LIN {X 0,Y 418.948,Z 202.65,A -85,B 0,C 180,E1 -10203.452,E2 -10203.452} C_VEL
LIN {X 0,Y 418.263,Z 200.109,A -85,B 0,C 180,E1 -10203.965,E2 -10203.965} C_VEL
LIN {X 0,Y 418.238,Z 200.015,A -85,B 0,C 180,E1 -10207.224,E2 -10207.224} C_VEL
LIN {X 0,Y 418.241,Z 199.978,A -85,B 0,C 180,E1 -10209.683,E2 -10209.683} C_VEL
LIN {X 0,Y 418.228,Z 200.013,A -85,B 0,C 180,E1 -10212.321,E2 -10212.321} C_VEL
LIN {X 0,Y 418.234,Z 200.009,A -85,B 0,C 180,E1 -10215.109,E2 -10215.109} C_VEL
LIN {X 0,Y 418.238,Z 200.002,A -85,B 0,C 180,E1 -10217.767,E2 -10217.767} C_VEL
LIN {X 0,Y 418.256,Z 200.011,A -85,B 0,C 180,E1 -10220.618,E2 -10220.618} C_VEL
LIN {X 0,Y 418.241,Z 200.01,A -85,B 0,C 180,E1 -10223.976,E2 -10223.976} C_VEL
LIN {X 0,Y 418.255,Z 199.993,A -85,B 0,C 180,E1 -10227.156,E2 -10227.156} C_VEL
LIN {X 0,Y 418.266,Z 200.006,A -85,B 0,C 180,E1 -10230.895,E2 -10230.895} C_VEL
LIN {X 0,Y 418.265,Z 199.989,A -85,B 0,C 180,E1 -10234.096,E2 -10234.096} C_VEL
LIN {X 0,Y 418.235,Z 200.01,A -85,B 0,C 180,E1 -10237.264,E2 -10237.264} C_VEL
LIN {X 0,Y 418.281,Z 200.008,A -85,B 0,C 180,E1 -10240.364,E2 -10240.364} C_VEL
LIN {X 0,Y 418.315,Z 199.999,A -85,B 0,C 180,E1 -10243.405,E2 -10243.405} C_VEL
LIN {X 0,Y 418.344,Z 199.994,A -85,B 0,C 180,E1 -10246.999,E2 -10246.999} C_VEL
LIN {X 0,Y 418.338,Z 199.995,A -85,B 0,C 180,E1 -10250.329,E2 -10250.329} C_VEL
LIN {X 0,Y 418.49,Z 199.98,A -85,B 0,C 180,E1 -10253.249,E2 -10253.249} C_VEL
LIN {X 0,Y 418.337,Z 199.993,A -85,B 0,C 180,E1 -10255.182,E2 -10255.182} C_VEL
LIN {X 0,Y 418.54,Z 199.968,A -85,B 0,C 180,E1 -10258.076,E2 -10258.076} C_VEL
LIN {X 0,Y 418.668,Z 199.959,A -85,B 0,C 180,E1 -10260,E2 -10260} C_VEL
LIN {X 0,Y 418.499,Z 199.974,A -85,B 0,C 180,E1 -10262.888,E2 -10262.888} C_VEL
LIN {X 0,Y 418.491,Z 199.977,A -85,B 0,C 180,E1 -10266.751,E2 -10266.751} C_VEL
LIN {X 0,Y 418.398,Z 199.988,A -85,B 0,C 180,E1 -10268.695,E2 -10268.695} C_VEL
LIN {X 0,Y 418.313,Z 199.997,A -85,B 0,C 180,E1 -10271.631,E2 -10271.631} C_VEL
LIN {X 0,Y 418.302,Z 200.003,A -85,B 0,C 180,E1 -10274.597,E2 -10274.597} C_VEL
LIN {X 0,Y 418.286,Z 200.007,A -85,B 0,C 180,E1 -10277.604,E2 -10277.604} C_VEL
LIN {X 0,Y 418.248,Z 200.005,A -85,B 0,C 180,E1 -10280.663,E2 -10280.663} C_VEL
LIN {X 0,Y 418.286,Z 200.001,A -85,B 0,C 180,E1 -10283.781,E2 -10283.781} C_VEL
LIN {X 0,Y 418.309,Z 199.995,A -85,B 0,C 180,E1 -10287.071,E2 -10287.071} C_VEL
LIN {X 0,Y 418.243,Z 200.002,A -85,B 0,C 180,E1 -10290.272,E2 -10290.272} C_VEL
LIN {X 0,Y 418.248,Z 200.002,A -85,B 0,C 180,E1 -10293.677,E2 -10293.677} C_VEL
LIN {X 0,Y 418.245,Z 200.012,A -85,B 0,C 180,E1 -10297.224,E2 -10297.224} C_VEL
LIN {X 0,Y 418.245,Z 199.997,A -85,B 0,C 180,E1 -10299.683,E2 -10299.683} C_VEL
LIN {X 0,Y 418.229,Z 200.016,A -85,B 0,C 180,E1 -10302.321,E2 -10302.321} C_VEL
LIN {X 0,Y 418.236,Z 200.01,A -85,B 0,C 180,E1 -10305.109,E2 -10305.109} C_VEL
LIN {X 0,Y 418.241,Z 200.003,A -85,B 0,C 180,E1 -10307.767,E2 -10307.767} C_VEL
LIN {X 0,Y 418.257,Z 200.007,A -85,B 0,C 180,E1 -10311.559,E2 -10311.559} C_VEL
LIN {X 0,Y 418.261,Z 200.008,A -85,B 0,C 180,E1 -10315.159,E2 -10315.159} C_VEL
LIN {X 0,Y 418.264,Z 200.161,A -85,B 0,C 180,E1 -10317.936,E2 -10317.936} C_VEL
LIN {X 0,Y 421.61,Z 212.936,A -85,B 0,C 180,E1 -10320.666,E2 -10320.666} C_VEL
LIN {X 0,Y 424.492,Z 225.433,A -85,B 0,C 180,E1 -10323.183,E2 -10323.183} C_VEL
LIN {X 0,Y 424.056,Z 232.827,A -85,B 0,C 180,E1 -10324.475,E2 -10324.475} C_VEL
LIN {X 0,Y 423.178,Z 244.55,A -85,B 0,C 180,E1 -10326.446,E2 -10326.446} C_VEL
LIN {X 0,Y 428.61,Z 271.164,A -85,B 0,C 180,E1 -10327.259,E2 -10327.259} C_VEL
LIN {X 0,Y 427.159,Z 386.676,A -85,B 0,C 180,E1 -10329.126,E2 -10329.126} C_VEL
LIN {X 0,Y 426.648,Z 400.992,A -85,B 0,C 180,E1 -10329.541,E2 -10329.541} C_VEL
LIN {X 0,Y 426.043,Z 413.972,A -85,B 0,C 180,E1 -10330.098,E2 -10330.098} C_VEL
LIN {X 0,Y 425.195,Z 426.696,A -85,B 0,C 180,E1 -10330.821,E2 -10330.821} C_VEL
LIN {X 0,Y 424.185,Z 439.707,A -85,B 0,C 180,E1 -10331.776,E2 -10331.776} C_VEL
LIN {X 0,Y 423.012,Z 451.477,A -85,B 0,C 180,E1 -10332.848,E2 -10332.848} C_VEL
LIN {X 0,Y 422.014,Z 462.206,A -85,B 0,C 180,E1 -10334.051,E2 -10334.051} C_VEL
LIN {X 0,Y 421.84,Z 463.782,A -85,B 0,C 180,E1 -10334.248,E2 -10334.248} C_VEL
LIN {X 0,Y 420.765,Z 468.085,A -85,B 0,C 180,E1 -10334.781,E2 -10334.781} C_VEL
LIN {X 0,Y 417.353,Z 474.899,A -85,B 0,C 180,E1 -10335.649,E2 -10335.649} C_VEL
LIN {X 0,Y 413.895,Z 481.189,A -85,B 0,C 180,E1 -10336.592,E2 -10336.592} C_VEL
LIN {X 0,Y 412.765,Z 484.669,A -85,B 0,C 180,E1 -10337.236,E2 -10337.236} C_VEL
LIN {X 0,Y 411.874,Z 492.436,A -85,B 0,C 180,E1 -10338.932,E2 -10338.932} C_VEL
LIN {X 0,Y 411.196,Z 498.815,A -85,B 0,C 180,E1 -10340.655,E2 -10340.655} C_VEL
LIN {X 0,Y 410.701,Z 504.611,A -85,B 0,C 180,E1 -10342.675,E2 -10342.675} C_VEL
LIN {X 0,Y 410.463,Z 507.781,A -85,B 0,C 180,E1 -10344.103,E2 -10344.103} C_VEL
LIN {X 0,Y 410.21,Z 510.948,A -85,B 0,C 180,E1 -10346.07,E2 -10346.07} C_VEL
LIN {X 0,Y 410.075,Z 512.822,A -85,B 0,C 180,E1 -10348.035,E2 -10348.035} C_VEL
LIN {X 0,Y 409.976,Z 513.463,A -85,B 0,C 180,E1 -10350,E2 -10350} C_VEL
LIN {X 0,Y 410.065,Z 512.885,A -85,B 0,C 180,E1 -10351.964,E2 -10351.964} C_VEL
LIN {X 0,Y 410.187,Z 511.079,A -85,B 0,C 180,E1 -10353.929,E2 -10353.929} C_VEL
LIN {X 0,Y 410.456,Z 507.979,A -85,B 0,C 180,E1 -10355.896,E2 -10355.896} C_VEL
LIN {X 0,Y 410.733,Z 503.489,A -85,B 0,C 180,E1 -10357.867,E2 -10357.867} C_VEL
LIN {X 0,Y 411.326,Z 497.457,A -85,B 0,C 180,E1 -10359.837,E2 -10359.837} C_VEL
LIN {X 0,Y 412.044,Z 490.753,A -85,B 0,C 180,E1 -10361.561,E2 -10361.561} C_VEL
LIN {X 0,Y 413.022,Z 482.453,A -85,B 0,C 180,E1 -10363.28,E2 -10363.28} C_VEL
LIN {X 0,Y 413.928,Z 473.814,A -85,B 0,C 180,E1 -10364.754,E2 -10364.754} C_VEL
LIN {X 0,Y 415.113,Z 463.352,A -85,B 0,C 180,E1 -10366.221,E2 -10366.221} C_VEL
LIN {X 0,Y 416.199,Z 452.792,A -85,B 0,C 180,E1 -10367.441,E2 -10367.441} C_VEL
LIN {X 0,Y 417.416,Z 441.262,A -85,B 0,C 180,E1 -10368.529,E2 -10368.529} C_VEL
LIN {X 0,Y 418.401,Z 428.579,A -85,B 0,C 180,E1 -10369.502,E2 -10369.502} C_VEL
LIN {X 0,Y 419.385,Z 414.919,A -85,B 0,C 180,E1 -10370.31,E2 -10370.31} C_VEL
LIN {X 0,Y 420.082,Z 401.003,A -85,B 0,C 180,E1 -10370.92,E2 -10370.92} C_VEL
LIN {X 0,Y 420.614,Z 386.556,A -85,B 0,C 180,E1 -10371.342,E2 -10371.342} C_VEL
LIN {X 0,Y 422.183,Z 272.349,A -85,B 0,C 180,E1 -10373.21,E2 -10373.21} C_VEL
LIN {X 0,Y 416.52,Z 244.696,A -85,B 0,C 180,E1 -10374.076,E2 -10374.076} C_VEL
LIN {X 0,Y 416.759,Z 240.683,A -85,B 0,C 180,E1 -10374.716,E2 -10374.716} C_VEL
LIN {X 0,Y 417.817,Z 228.064,A -85,B 0,C 180,E1 -10376.937,E2 -10376.937} C_VEL
LIN {X 0,Y 414.837,Z 214.884,A -85,B 0,C 180,E1 -10379.622,E2 -10379.622} C_VEL
LIN {X 0,Y 411.239,Z 201.027,A -85,B 0,C 180,E1 -10382.638,E2 -10382.638} C_VEL
LIN {X 0,Y 411.198,Z 200.892,A -85,B 0,C 180,E1 -10385.528,E2 -10385.528} C_VEL
LIN {X 0,Y 411.216,Z 200.882,A -85,B 0,C 180,E1 -10389.223,E2 -10389.223} C_VEL
LIN {X 0,Y 411.179,Z 200.884,A -85,B 0,C 180,E1 -10392.695,E2 -10392.695} C_VEL
LIN {X 0,Y 411.165,Z 200.884,A -85,B 0,C 180,E1 -10395.88,E2 -10395.88} C_VEL
LIN {X 0,Y 411.16,Z 200.895,A -85,B 0,C 180,E1 -10398.771,E2 -10398.771} C_VEL
LIN {X 0,Y 411.192,Z 200.891,A -85,B 0,C 180,E1 -10402.026,E2 -10402.026} C_VEL
LIN {X 0,Y 411.201,Z 200.874,A -85,B 0,C 180,E1 -10405.666,E2 -10405.666} C_VEL
LIN {X 0,Y 411.193,Z 200.887,A -85,B 0,C 180,E1 -10409.152,E2 -10409.152} C_VEL
LIN {X 0,Y 411.254,Z 200.868,A -85,B 0,C 180,E1 -10412.522,E2 -10412.522} C_VEL
LIN {X 0,Y 411.221,Z 200.881,A -85,B 0,C 180,E1 -10415.784,E2 -10415.784} C_VEL
LIN {X 0,Y 411.19,Z 200.889,A -85,B 0,C 180,E1 -10418.965,E2 -10418.965} C_VEL
LIN {X 0,Y 411.246,Z 200.881,A -85,B 0,C 180,E1 -10422.084,E2 -10422.084} C_VEL
LIN {X 0,Y 411.256,Z 200.883,A -85,B 0,C 180,E1 -10425.147,E2 -10425.147} C_VEL
LIN {X 0,Y 411.277,Z 200.873,A -85,B 0,C 180,E1 -10428.167,E2 -10428.167} C_VEL
LIN {X 0,Y 411.475,Z 200.85,A -85,B 0,C 180,E1 -10432.146,E2 -10432.146} C_VEL
LIN {X 0,Y 411.468,Z 200.854,A -85,B 0,C 180,E1 -10434.118,E2 -10434.118} C_VEL
LIN {X 0,Y 411.507,Z 200.847,A -85,B 0,C 180,E1 -10438.042,E2 -10438.042} C_VEL
LIN {X 0,Y 411.635,Z 200.835,A -85,B 0,C 180,E1 -10440,E2 -10440} C_VEL
LIN {X 0,Y 411.459,Z 200.855,A -85,B 0,C 180,E1 -10442.937,E2 -10442.937} C_VEL
LIN {X 0,Y 411.453,Z 200.856,A -85,B 0,C 180,E1 -10446.867,E2 -10446.867} C_VEL
LIN {X 0,Y 411.286,Z 200.873,A -85,B 0,C 180,E1 -10449.839,E2 -10449.839} C_VEL
LIN {X 0,Y 411.298,Z 200.872,A -85,B 0,C 180,E1 -10453.104,E2 -10453.104} C_VEL
LIN {X 0,Y 411.25,Z 200.878,A -85,B 0,C 180,E1 -10456.889,E2 -10456.889} C_VEL
LIN {X 0,Y 411.223,Z 200.887,A -85,B 0,C 180,E1 -10459.987,E2 -10459.987} C_VEL
LIN {X 0,Y 411.196,Z 200.888,A -85,B 0,C 180,E1 -10463.148,E2 -10463.148} C_VEL
LIN {X 0,Y 411.231,Z 200.862,A -85,B 0,C 180,E1 -10466.381,E2 -10466.381} C_VEL
LIN {X 0,Y 411.194,Z 200.893,A -85,B 0,C 180,E1 -10469.713,E2 -10469.713} C_VEL
LIN {X 0,Y 411.2,Z 200.872,A -85,B 0,C 180,E1 -10473.156,E2 -10473.156} C_VEL
LIN {X 0,Y 411.187,Z 200.885,A -85,B 0,C 180,E1 -10476.553,E2 -10476.553} C_VEL
LIN {X 0,Y 411.212,Z 200.89,A -85,B 0,C 180,E1 -10479.729,E2 -10479.729} C_VEL
LIN {X 0,Y 411.168,Z 200.889,A -85,B 0,C 180,E1 -10483.134,E2 -10483.134} C_VEL
LIN {X 0,Y 411.163,Z 200.887,A -85,B 0,C 180,E1 -10485.882,E2 -10485.882} C_VEL
LIN {X 0,Y 411.158,Z 200.874,A -85,B 0,C 180,E1 -10488.772,E2 -10488.772} C_VEL
LIN {X 0,Y 411.186,Z 200.884,A -85,B 0,C 180,E1 -10492.026,E2 -10492.026} C_VEL
LIN {X 0,Y 411.246,Z 201.009,A -85,B 0,C 180,E1 -10495.536,E2 -10495.536} C_VEL
LIN {X 0,Y 415.16,Z 214.888,A -85,B 0,C 180,E1 -10498.206,E2 -10498.206} C_VEL
LIN {X 0,Y 418.193,Z 226.388,A -85,B 0,C 180,E1 -10500.281,E2 -10500.281} C_VEL
LIN {X 0,Y 419.41,Z 231.713,A -85,B 0,C 180,E1 -10501.2,E2 -10501.2} C_VEL
LIN {X 0,Y 418.207,Z 245.027,A -85,B 0,C 180,E1 -10503.147,E2 -10503.147} C_VEL
LIN {X 0,Y 422.74,Z 272.159,A -85,B 0,C 180,E1 -10503.981,E2 -10503.981} C_VEL
LIN {X 0,Y 420.155,Z 407.504,A -85,B 0,C 180,E1 -10506.463,E2 -10506.463} C_VEL
LIN {X 0,Y 419.399,Z 423.23,A -85,B 0,C 180,E1 -10506.94,E2 -10506.94} C_VEL
LIN {X 0,Y 418.546,Z 437.915,A -85,B 0,C 180,E1 -10507.585,E2 -10507.585} C_VEL
LIN {X 0,Y 417.477,Z 451.995,A -85,B 0,C 180,E1 -10508.393,E2 -10508.393} C_VEL
LIN {X 0,Y 416.343,Z 465.452,A -85,B 0,C 180,E1 -10509.368,E2 -10509.368} C_VEL
LIN {X 0,Y 415.216,Z 477.877,A -85,B 0,C 180,E1 -10510.471,E2 -10510.471} C_VEL
LIN {X 0,Y 414.074,Z 490.391,A -85,B 0,C 180,E1 -10511.811,E2 -10511.811} C_VEL
LIN {X 0,Y 413.093,Z 501.14,A -85,B 0,C 180,E1 -10513.189,E2 -10513.189} C_VEL
LIN {X 0,Y 412.123,Z 510.953,A -85,B 0,C 180,E1 -10514.674,E2 -10514.674} C_VEL
LIN {X 0,Y 411.31,Z 520.71,A -85,B 0,C 180,E1 -10516.437,E2 -10516.437} C_VEL
LIN {X 0,Y 410.753,Z 528.58,A -85,B 0,C 180,E1 -10518.152,E2 -10518.152} C_VEL
LIN {X 0,Y 410.429,Z 534.358,A -85,B 0,C 180,E1 -10519.643,E2 -10519.643} C_VEL
LIN {X 0,Y 410.127,Z 540.599,A -85,B 0,C 180,E1 -10521.625,E2 -10521.625} C_VEL
LIN {X 0,Y 410.046,Z 544.283,A -85,B 0,C 180,E1 -10523.11,E2 -10523.11} C_VEL
LIN {X 0,Y 409.971,Z 548.051,A -85,B 0,C 180,E1 -10525.083,E2 -10525.083} C_VEL
LIN {X 0,Y 409.984,Z 550.533,A -85,B 0,C 180,E1 -10527.053,E2 -10527.053} C_VEL
LIN {X 0,Y 409.975,Z 551.778,A -85,B 0,C 180,E1 -10529.018,E2 -10529.018} C_VEL
LIN {X 0,Y 409.976,Z 551.776,A -85,B 0,C 180,E1 -10530.983,E2 -10530.983} C_VEL
LIN {X 0,Y 409.985,Z 550.524,A -85,B 0,C 180,E1 -10532.948,E2 -10532.948} C_VEL
LIN {X 0,Y 410,Z 548.04,A -85,B 0,C 180,E1 -10534.917,E2 -10534.917} C_VEL
LIN {X 0,Y 410.067,Z 544.273,A -85,B 0,C 180,E1 -10536.891,E2 -10536.891} C_VEL
LIN {X 0,Y 410.193,Z 539.132,A -85,B 0,C 180,E1 -10538.871,E2 -10538.871} C_VEL
LIN {X 0,Y 410.542,Z 532.489,A -85,B 0,C 180,E1 -10540.854,E2 -10540.854} C_VEL
LIN {X 0,Y 411.093,Z 524.16,A -85,B 0,C 180,E1 -10542.841,E2 -10542.841} C_VEL
LIN {X 0,Y 411.781,Z 515.261,A -85,B 0,C 180,E1 -10544.581,E2 -10544.581} C_VEL
LIN {X 0,Y 412.706,Z 504.537,A -85,B 0,C 180,E1 -10546.319,E2 -10546.319} C_VEL
LIN {X 0,Y 413.76,Z 493.517,A -85,B 0,C 180,E1 -10547.803,E2 -10547.803} C_VEL
LIN {X 0,Y 414.841,Z 481.467,A -85,B 0,C 180,E1 -10549.162,E2 -10549.162} C_VEL
LIN {X 0,Y 415.92,Z 469.712,A -85,B 0,C 180,E1 -10550.267,E2 -10550.267} C_VEL
LIN {X 0,Y 417.161,Z 455.436,A -85,B 0,C 180,E1 -10551.366,E2 -10551.366} C_VEL
LIN {X 0,Y 418.232,Z 441.838,A -85,B 0,C 180,E1 -10552.2,E2 -10552.2} C_VEL
LIN {X 0,Y 419.174,Z 426.827,A -85,B 0,C 180,E1 -10552.911,E2 -10552.911} C_VEL
LIN {X 0,Y 419.925,Z 411.687,A -85,B 0,C 180,E1 -10553.421,E2 -10553.421} C_VEL
LIN {X 0,Y 420.517,Z 391.478,A -85,B 0,C 180,E1 -10553.844,E2 -10553.844} C_VEL
LIN {X 0,Y 422.719,Z 272.152,A -85,B 0,C 180,E1 -10556.011,E2 -10556.011} C_VEL
LIN {X 0,Y 418.252,Z 245.233,A -85,B 0,C 180,E1 -10556.826,E2 -10556.826} C_VEL
LIN {X 0,Y 419.408,Z 231.698,A -85,B 0,C 180,E1 -10558.801,E2 -10558.801} C_VEL
LIN {X 0,Y 416.321,Z 219.072,A -85,B 0,C 180,E1 -10561.021,E2 -10561.021} C_VEL
LIN {X 0,Y 412.289,Z 204.82,A -85,B 0,C 180,E1 -10563.681,E2 -10563.681} C_VEL
LIN {X 0,Y 411.246,Z 200.982,A -85,B 0,C 180,E1 -10564.465,E2 -10564.465} C_VEL
LIN {X 0,Y 411.198,Z 200.877,A -85,B 0,C 180,E1 -10568.168,E2 -10568.168} C_VEL
LIN {X 0,Y 411.162,Z 200.874,A -85,B 0,C 180,E1 -10571.228,E2 -10571.228} C_VEL
LIN {X 0,Y 411.174,Z 200.885,A -85,B 0,C 180,E1 -10574.49,E2 -10574.49} C_VEL
LIN {X 0,Y 411.175,Z 200.882,A -85,B 0,C 180,E1 -10578.195,E2 -10578.195} C_VEL
LIN {X 0,Y 411.22,Z 200.885,A -85,B 0,C 180,E1 -10580.776,E2 -10580.776} C_VEL
LIN {X 0,Y 411.196,Z 200.893,A -85,B 0,C 180,E1 -10584.471,E2 -10584.471} C_VEL
LIN {X 0,Y 411.205,Z 200.872,A -85,B 0,C 180,E1 -10586.873,E2 -10586.873} C_VEL
LIN {X 0,Y 411.231,Z 200.885,A -85,B 0,C 180,E1 -10590.644,E2 -10590.644} C_VEL
LIN {X 0,Y 411.234,Z 200.861,A -85,B 0,C 180,E1 -10593.619,E2 -10593.619} C_VEL
LIN {X 0,Y 411.2,Z 200.888,A -85,B 0,C 180,E1 -10596.852,E2 -10596.852} C_VEL
LIN {X 0,Y 411.213,Z 200.889,A -85,B 0,C 180,E1 -10600.05,E2 -10600.05} C_VEL
LIN {X 0,Y 411.261,Z 200.877,A -85,B 0,C 180,E1 -10603.131,E2 -10603.131} C_VEL
LIN {X 0,Y 411.303,Z 200.871,A -85,B 0,C 180,E1 -10606.896,E2 -10606.896} C_VEL
LIN {X 0,Y 411.29,Z 200.872,A -85,B 0,C 180,E1 -10610.161,E2 -10610.161} C_VEL
LIN {X 0,Y 411.454,Z 200.856,A -85,B 0,C 180,E1 -10613.133,E2 -10613.133} C_VEL
LIN {X 0,Y 411.308,Z 200.868,A -85,B 0,C 180,E1 -10615.099,E2 -10615.099} C_VEL
LIN {X 0,Y 411.509,Z 200.844,A -85,B 0,C 180,E1 -10618.043,E2 -10618.043} C_VEL
LIN {X 0,Y 411.637,Z 200.835,A -85,B 0,C 180,E1 -10620,E2 -10620} C_VEL
LIN {X 0,Y 411.456,Z 200.852,A -85,B 0,C 180,E1 -10622.937,E2 -10622.937} C_VEL
LIN {X 0,Y 411.458,Z 200.854,A -85,B 0,C 180,E1 -10626.867,E2 -10626.867} C_VEL
LIN {X 0,Y 411.352,Z 200.866,A -85,B 0,C 180,E1 -10628.845,E2 -10628.845} C_VEL
LIN {X 0,Y 411.282,Z 200.872,A -85,B 0,C 180,E1 -10631.833,E2 -10631.833} C_VEL
LIN {X 0,Y 411.259,Z 200.882,A -85,B 0,C 180,E1 -10634.853,E2 -10634.853} C_VEL
LIN {X 0,Y 411.251,Z 200.881,A -85,B 0,C 180,E1 -10637.915,E2 -10637.915} C_VEL
LIN {X 0,Y 411.195,Z 200.888,A -85,B 0,C 180,E1 -10641.034,E2 -10641.034} C_VEL
LIN {X 0,Y 411.225,Z 200.88,A -85,B 0,C 180,E1 -10644.216,E2 -10644.216} C_VEL
LIN {X 0,Y 411.258,Z 200.868,A -85,B 0,C 180,E1 -10647.478,E2 -10647.478} C_VEL
LIN {X 0,Y 411.188,Z 200.886,A -85,B 0,C 180,E1 -10650.848,E2 -10650.848} C_VEL
LIN {X 0,Y 411.206,Z 200.874,A -85,B 0,C 180,E1 -10654.334,E2 -10654.334} C_VEL
LIN {X 0,Y 411.196,Z 200.889,A -85,B 0,C 180,E1 -10657.974,E2 -10657.974} C_VEL
LIN {X 0,Y 411.164,Z 200.893,A -85,B 0,C 180,E1 -10661.229,E2 -10661.229} C_VEL
LIN {X 0,Y 411.176,Z 200.883,A -85,B 0,C 180,E1 -10664.491,E2 -10664.491} C_VEL
LIN {X 0,Y 411.178,Z 200.884,A -85,B 0,C 180,E1 -10668.195,E2 -10668.195} C_VEL
LIN {X 0,Y 411.22,Z 200.881,A -85,B 0,C 180,E1 -10670.776,E2 -10670.776} C_VEL
LIN {X 0,Y 411.2,Z 200.891,A -85,B 0,C 180,E1 -10674.472,E2 -10674.472} C_VEL
LIN {X 0,Y 411.231,Z 201.077,A -85,B 0,C 180,E1 -10677.484,E2 -10677.484} C_VEL
LIN {X 0,Y 414.151,Z 212.297,A -85,B 0,C 180,E1 -10679.935,E2 -10679.935} C_VEL
LIN {X 0,Y 416.984,Z 224.123,A -85,B 0,C 180,E1 -10682.387,E2 -10682.387} C_VEL
LIN {X 0,Y 417.795,Z 228.696,A -85,B 0,C 180,E1 -10683.289,E2 -10683.289} C_VEL
LIN {X 0,Y 416.48,Z 244.569,A -85,B 0,C 180,E1 -10686.016,E2 -10686.016} C_VEL
LIN {X 0,Y 422.058,Z 271.648,A -85,B 0,C 180,E1 -10686.867,E2 -10686.867} C_VEL
LIN {X 0,Y 420.622,Z 386.454,A -85,B 0,C 180,E1 -10688.754,E2 -10688.754} C_VEL
LIN {X 0,Y 420.091,Z 400.957,A -85,B 0,C 180,E1 -10689.175,E2 -10689.175} C_VEL
LIN {X 0,Y 419.399,Z 414.888,A -85,B 0,C 180,E1 -10689.787,E2 -10689.787} C_VEL
LIN {X 0,Y 418.519,Z 427.216,A -85,B 0,C 180,E1 -10690.503,E2 -10690.503} C_VEL
LIN {X 0,Y 417.473,Z 440.174,A -85,B 0,C 180,E1 -10691.473,E2 -10691.473} C_VEL
LIN {X 0,Y 416.257,Z 451.907,A -85,B 0,C 180,E1 -10692.561,E2 -10692.561} C_VEL
LIN {X 0,Y 415.192,Z 462.612,A -85,B 0,C 180,E1 -10693.782,E2 -10693.782} C_VEL
LIN {X 0,Y 413.989,Z 473.195,A -85,B 0,C 180,E1 -10695.247,E2 -10695.247} C_VEL
LIN {X 0,Y 413.118,Z 481.937,A -85,B 0,C 180,E1 -10696.723,E2 -10696.723} C_VEL
LIN {X 0,Y 412.765,Z 484.669,A -85,B 0,C 180,E1 -10697.236,E2 -10697.236} C_VEL
LIN {X 0,Y 411.645,Z 488.055,A -85,B 0,C 180,E1 -10697.901,E2 -10697.901} C_VEL
LIN {X 0,Y 408.234,Z 493.211,A -85,B 0,C 180,E1 -10698.985,E2 -10698.985} C_VEL
LIN {X 0,Y 404.961,Z 497.856,A -85,B 0,C 180,E1 -10700.126,E2 -10700.126} C_VEL
LIN {X 0,Y 404.063,Z 500.337,A -85,B 0,C 180,E1 -10700.87,E2 -10700.87} C_VEL
LIN {X 0,Y 403.663,Z 504.834,A -85,B 0,C 180,E1 -10702.497,E2 -10702.497} C_VEL
LIN {X 0,Y 403.421,Z 508.12,A -85,B 0,C 180,E1 -10704,E2 -10704} C_VEL
LIN {X 0,Y 403.121,Z 511.284,A -85,B 0,C 180,E1 -10706.001,E2 -10706.001} C_VEL
LIN {X 0,Y 403.006,Z 513.154,A -85,B 0,C 180,E1 -10708.001,E2 -10708.001} C_VEL
LIN {X 0,Y 402.898,Z 513.795,A -85,B 0,C 180,E1 -10710,E2 -10710} C_VEL
LIN {X 0,Y 402.997,Z 513.217,A -85,B 0,C 180,E1 -10711.998,E2 -10711.998} C_VEL
LIN {X 0,Y 403.125,Z 512.467,A -85,B 0,C 180,E1 -10712.998,E2 -10712.998} C_VEL
LIN {X 0,Y 403.156,Z 510.035,A -85,B 0,C 180,E1 -10715,E2 -10715} C_VEL
LIN {X 0,Y 403.566,Z 506.254,A -85,B 0,C 180,E1 -10717.001,E2 -10717.001} C_VEL
LIN {X 0,Y 404.001,Z 501.021,A -85,B 0,C 180,E1 -10719.007,E2 -10719.007} C_VEL
LIN {X 0,Y 404.756,Z 494.15,A -85,B 0,C 180,E1 -10721.011,E2 -10721.011} C_VEL
LIN {X 0,Y 405.625,Z 486.583,A -85,B 0,C 180,E1 -10722.762,E2 -10722.762} C_VEL
LIN {X 0,Y 406.65,Z 477.932,A -85,B 0,C 180,E1 -10724.393,E2 -10724.393} C_VEL
LIN {X 0,Y 407.658,Z 469.228,A -85,B 0,C 180,E1 -10725.755,E2 -10725.755} C_VEL
LIN {X 0,Y 408.905,Z 458.721,A -85,B 0,C 180,E1 -10727.117,E2 -10727.117} C_VEL
LIN {X 0,Y 410.085,Z 447.116,A -85,B 0,C 180,E1 -10728.355,E2 -10728.355} C_VEL
LIN {X 0,Y 411.244,Z 435.757,A -85,B 0,C 180,E1 -10729.336,E2 -10729.336} C_VEL
LIN {X 0,Y 412.21,Z 423.673,A -85,B 0,C 180,E1 -10730.181,E2 -10730.181} C_VEL
LIN {X 0,Y 413.102,Z 409.749,A -85,B 0,C 180,E1 -10730.932,E2 -10730.932} C_VEL
LIN {X 0,Y 413.733,Z 396.35,A -85,B 0,C 180,E1 -10731.453,E2 -10731.453} C_VEL
LIN {X 0,Y 414.151,Z 383.076,A -85,B 0,C 180,E1 -10731.79,E2 -10731.79} C_VEL
LIN {X 0,Y 415.75,Z 273.499,A -85,B 0,C 180,E1 -10733.597,E2 -10733.597} C_VEL
LIN {X 0,Y 410.069,Z 245.992,A -85,B 0,C 180,E1 -10734.467,E2 -10734.467} C_VEL
LIN {X 0,Y 409.807,Z 244.124,A -85,B 0,C 180,E1 -10734.578,E2 -10734.578} C_VEL
LIN {X 0,Y 411.051,Z 230.507,A -85,B 0,C 180,E1 -10736.99,E2 -10736.99} C_VEL
LIN {X 0,Y 408.624,Z 219.018,A -85,B 0,C 180,E1 -10739.351,E2 -10739.351} C_VEL
LIN {X 0,Y 405.098,Z 205.35,A -85,B 0,C 180,E1 -10742.323,E2 -10742.323} C_VEL
LIN {X 0,Y 404.175,Z 201.859,A -85,B 0,C 180,E1 -10743.152,E2 -10743.152} C_VEL
LIN {X 0,Y 404.142,Z 201.763,A -85,B 0,C 180,E1 -10746.245,E2 -10746.245} C_VEL
LIN {X 0,Y 404.154,Z 201.763,A -85,B 0,C 180,E1 -10748.756,E2 -10748.756} C_VEL
LIN {X 0,Y 404.12,Z 201.766,A -85,B 0,C 180,E1 -10751.599,E2 -10751.599} C_VEL
LIN {X 0,Y 404.144,Z 201.767,A -85,B 0,C 180,E1 -10754.521,E2 -10754.521} C_VEL
LIN {X 0,Y 404.133,Z 201.768,A -85,B 0,C 180,E1 -10757.295,E2 -10757.295} C_VEL
LIN {X 0,Y 404.165,Z 201.751,A -85,B 0,C 180,E1 -10759.955,E2 -10759.955} C_VEL
LIN {X 0,Y 404.135,Z 201.772,A -85,B 0,C 180,E1 -10763.124,E2 -10763.124} C_VEL
LIN {X 0,Y 404.14,Z 201.758,A -85,B 0,C 180,E1 -10766.187,E2 -10766.187} C_VEL
LIN {X 0,Y 404.148,Z 201.758,A -85,B 0,C 180,E1 -10769.715,E2 -10769.715} C_VEL
LIN {X 0,Y 404.19,Z 201.754,A -85,B 0,C 180,E1 -10773.122,E2 -10773.122} C_VEL
LIN {X 0,Y 404.171,Z 201.762,A -85,B 0,C 180,E1 -10775.334,E2 -10775.334} C_VEL
LIN {X 0,Y 404.132,Z 201.77,A -85,B 0,C 180,E1 -10778.58,E2 -10778.58} C_VEL
LIN {X 0,Y 404.204,Z 201.758,A -85,B 0,C 180,E1 -10781.761,E2 -10781.761} C_VEL
LIN {X 0,Y 404.201,Z 201.758,A -85,B 0,C 180,E1 -10784.882,E2 -10784.882} C_VEL
LIN {X 0,Y 404.25,Z 201.748,A -85,B 0,C 180,E1 -10787.958,E2 -10787.958} C_VEL
LIN {X 0,Y 404.427,Z 201.728,A -85,B 0,C 180,E1 -10792.099,E2 -10792.099} C_VEL
LIN {X 0,Y 404.417,Z 201.731,A -85,B 0,C 180,E1 -10794.015,E2 -10794.015} C_VEL
LIN {X 0,Y 404.476,Z 201.722,A -85,B 0,C 180,E1 -10798.008,E2 -10798.008} C_VEL
LIN {X 0,Y 404.604,Z 201.711,A -85,B 0,C 180,E1 -10800,E2 -10800} C_VEL
LIN {X 0,Y 404.416,Z 201.733,A -85,B 0,C 180,E1 -10802.988,E2 -10802.988} C_VEL
LIN {X 0,Y 404.404,Z 201.734,A -85,B 0,C 180,E1 -10806.987,E2 -10806.987} C_VEL
LIN {X 0,Y 404.251,Z 201.749,A -85,B 0,C 180,E1 -10810.012,E2 -10810.012} C_VEL
LIN {X 0,Y 404.259,Z 201.748,A -85,B 0,C 180,E1 -10813.211,E2 -10813.211} C_VEL
LIN {X 0,Y 404.209,Z 201.755,A -85,B 0,C 180,E1 -10817.007,E2 -10817.007} C_VEL
LIN {X 0,Y 404.157,Z 201.763,A -85,B 0,C 180,E1 -10820.352,E2 -10820.352} C_VEL
LIN {X 0,Y 404.163,Z 201.768,A -85,B 0,C 180,E1 -10823.575,E2 -10823.575} C_VEL
LIN {X 0,Y 404.177,Z 201.744,A -85,B 0,C 180,E1 -10825.767,E2 -10825.767} C_VEL
LIN {X 0,Y 404.189,Z 201.752,A -85,B 0,C 180,E1 -10828,E2 -10828} C_VEL
LIN {X 0,Y 404.133,Z 201.756,A -85,B 0,C 180,E1 -10831.558,E2 -10831.558} C_VEL
LIN {X 0,Y 404.179,Z 201.763,A -85,B 0,C 180,E1 -10835.017,E2 -10835.017} C_VEL
LIN {X 0,Y 404.151,Z 201.761,A -85,B 0,C 180,E1 -10838.757,E2 -10838.757} C_VEL
LIN {X 0,Y 404.117,Z 201.761,A -85,B 0,C 180,E1 -10841.6,E2 -10841.6} C_VEL
LIN {X 0,Y 404.14,Z 201.768,A -85,B 0,C 180,E1 -10844.523,E2 -10844.523} C_VEL
LIN {X 0,Y 404.131,Z 201.773,A -85,B 0,C 180,E1 -10847.296,E2 -10847.296} C_VEL
LIN {X 0,Y 404.165,Z 201.73,A -85,B 0,C 180,E1 -10849.956,E2 -10849.956} C_VEL
LIN {X 0,Y 404.131,Z 201.765,A -85,B 0,C 180,E1 -10853.126,E2 -10853.126} C_VEL
LIN {X 0,Y 404.186,Z 201.933,A -85,B 0,C 180,E1 -10855.035,E2 -10855.035} C_VEL
LIN {X 0,Y 408.125,Z 215.592,A -85,B 0,C 180,E1 -10857.737,E2 -10857.737} C_VEL
LIN {X 0,Y 411.373,Z 227.977,A -85,B 0,C 180,E1 -10860.02,E2 -10860.02} C_VEL
LIN {X 0,Y 412.687,Z 233.627,A -85,B 0,C 180,E1 -10861.02,E2 -10861.02} C_VEL
LIN {X 0,Y 411.577,Z 245.037,A -85,B 0,C 180,E1 -10862.709,E2 -10862.709} C_VEL
LIN {X 0,Y 416.223,Z 272.495,A -85,B 0,C 180,E1 -10863.576,E2 -10863.576} C_VEL
LIN {X 0,Y 413.957,Z 393.97,A -85,B 0,C 180,E1 -10865.822,E2 -10865.822} C_VEL
LIN {X 0,Y 413.375,Z 412.135,A -85,B 0,C 180,E1 -10866.219,E2 -10866.219} C_VEL
LIN {X 0,Y 412.587,Z 427.051,A -85,B 0,C 180,E1 -10866.736,E2 -10866.736} C_VEL
LIN {X 0,Y 411.7,Z 440.535,A -85,B 0,C 180,E1 -10867.379,E2 -10867.379} C_VEL
LIN {X 0,Y 410.538,Z 455.044,A -85,B 0,C 180,E1 -10868.273,E2 -10868.273} C_VEL
LIN {X 0,Y 409.202,Z 469.332,A -85,B 0,C 180,E1 -10869.386,E2 -10869.386} C_VEL
LIN {X 0,Y 408.008,Z 482.292,A -85,B 0,C 180,E1 -10870.636,E2 -10870.636} C_VEL
LIN {X 0,Y 406.891,Z 493.161,A -85,B 0,C 180,E1 -10871.887,E2 -10871.887} C_VEL
LIN {X 0,Y 405.848,Z 504.196,A -85,B 0,C 180,E1 -10873.398,E2 -10873.398} C_VEL
LIN {X 0,Y 404.948,Z 513.533,A -85,B 0,C 180,E1 -10874.911,E2 -10874.911} C_VEL
LIN {X 0,Y 404.213,Z 521.735,A -85,B 0,C 180,E1 -10876.477,E2 -10876.477} C_VEL
LIN {X 0,Y 403.641,Z 530.289,A -85,B 0,C 180,E1 -10878.45,E2 -10878.45} C_VEL
LIN {X 0,Y 403.157,Z 537.319,A -85,B 0,C 180,E1 -10880.468,E2 -10880.468} C_VEL
LIN {X 0,Y 402.972,Z 542.826,A -85,B 0,C 180,E1 -10882.484,E2 -10882.484} C_VEL
LIN {X 0,Y 402.916,Z 545.994,A -85,B 0,C 180,E1 -10883.993,E2 -10883.993} C_VEL
LIN {X 0,Y 402.849,Z 549.113,A -85,B 0,C 180,E1 -10885.999,E2 -10885.999} C_VEL
LIN {X 0,Y 402.945,Z 550.978,A -85,B 0,C 180,E1 -10888.001,E2 -10888.001} C_VEL
LIN {X 0,Y 402.891,Z 551.606,A -85,B 0,C 180,E1 -10890,E2 -10890} C_VEL
LIN {X 0,Y 402.946,Z 550.972,A -85,B 0,C 180,E1 -10891.999,E2 -10891.999} C_VEL
LIN {X 0,Y 402.854,Z 549.1,A -85,B 0,C 180,E1 -10894.002,E2 -10894.002} C_VEL
LIN {X 0,Y 402.965,Z 545.983,A -85,B 0,C 180,E1 -10896.007,E2 -10896.007} C_VEL
LIN {X 0,Y 403.029,Z 541.536,A -85,B 0,C 180,E1 -10898.019,E2 -10898.019} C_VEL
LIN {X 0,Y 403.22,Z 535.652,A -85,B 0,C 180,E1 -10900.038,E2 -10900.038} C_VEL
LIN {X 0,Y 403.764,Z 528.189,A -85,B 0,C 180,E1 -10902.057,E2 -10902.057} C_VEL
LIN {X 0,Y 404.318,Z 520.302,A -85,B 0,C 180,E1 -10903.803,E2 -10903.803} C_VEL
LIN {X 0,Y 405.218,Z 510.529,A -85,B 0,C 180,E1 -10905.595,E2 -10905.595} C_VEL
LIN {X 0,Y 406.161,Z 500.684,A -85,B 0,C 180,E1 -10907.107,E2 -10907.107} C_VEL
LIN {X 0,Y 407.276,Z 488.972,A -85,B 0,C 180,E1 -10908.616,E2 -10908.616} C_VEL
LIN {X 0,Y 408.438,Z 477.355,A -85,B 0,C 180,E1 -10909.867,E2 -10909.867} C_VEL
LIN {X 0,Y 409.674,Z 464.868,A -85,B 0,C 180,E1 -10910.984,E2 -10910.984} C_VEL
LIN {X 0,Y 410.835,Z 451.333,A -85,B 0,C 180,E1 -10911.975,E2 -10911.975} C_VEL
LIN {X 0,Y 411.885,Z 437.239,A -85,B 0,C 180,E1 -10912.795,E2 -10912.795} C_VEL
LIN {X 0,Y 412.798,Z 422.296,A -85,B 0,C 180,E1 -10913.451,E2 -10913.451} C_VEL
LIN {X 0,Y 413.572,Z 407.375,A -85,B 0,C 180,E1 -10913.903,E2 -10913.903} C_VEL
LIN {X 0,Y 416.143,Z 281.51,A -85,B 0,C 180,E1 -10916.243,E2 -10916.243} C_VEL
LIN {X 0,Y 416.122,Z 272.091,A -85,B 0,C 180,E1 -10916.428,E2 -10916.428} C_VEL
LIN {X 0,Y 411.611,Z 245.018,A -85,B 0,C 180,E1 -10917.279,E2 -10917.279} C_VEL
LIN {X 0,Y 412.654,Z 233.604,A -85,B 0,C 180,E1 -10918.984,E2 -10918.984} C_VEL
LIN {X 0,Y 409.548,Z 220.88,A -85,B 0,C 180,E1 -10921.271,E2 -10921.271} C_VEL
LIN {X 0,Y 405.847,Z 207.701,A -85,B 0,C 180,E1 -10923.777,E2 -10923.777} C_VEL
LIN {X 0,Y 404.189,Z 201.889,A -85,B 0,C 180,E1 -10924.966,E2 -10924.966} C_VEL
LIN {X 0,Y 404.147,Z 201.741,A -85,B 0,C 180,E1 -10928.758,E2 -10928.758} C_VEL
LIN {X 0,Y 404.121,Z 201.758,A -85,B 0,C 180,E1 -10931.6,E2 -10931.6} C_VEL
LIN {X 0,Y 404.144,Z 201.76,A -85,B 0,C 180,E1 -10934.522,E2 -10934.522} C_VEL
LIN {X 0,Y 404.134,Z 201.761,A -85,B 0,C 180,E1 -10937.295,E2 -10937.295} C_VEL
LIN {X 0,Y 404.167,Z 201.766,A -85,B 0,C 180,E1 -10939.955,E2 -10939.955} C_VEL
LIN {X 0,Y 404.134,Z 201.762,A -85,B 0,C 180,E1 -10943.125,E2 -10943.125} C_VEL
LIN {X 0,Y 404.143,Z 201.761,A -85,B 0,C 180,E1 -10946.188,E2 -10946.188} C_VEL
LIN {X 0,Y 404.143,Z 201.765,A -85,B 0,C 180,E1 -10949.715,E2 -10949.715} C_VEL
LIN {X 0,Y 404.192,Z 201.739,A -85,B 0,C 180,E1 -10953.123,E2 -10953.123} C_VEL
LIN {X 0,Y 404.174,Z 201.757,A -85,B 0,C 180,E1 -10955.334,E2 -10955.334} C_VEL
LIN {X 0,Y 404.136,Z 201.765,A -85,B 0,C 180,E1 -10958.581,E2 -10958.581} C_VEL
LIN {X 0,Y 404.208,Z 201.757,A -85,B 0,C 180,E1 -10961.762,E2 -10961.762} C_VEL
LIN {X 0,Y 404.204,Z 201.757,A -85,B 0,C 180,E1 -10964.882,E2 -10964.882} C_VEL
LIN {X 0,Y 404.254,Z 201.757,A -85,B 0,C 180,E1 -10967.959,E2 -10967.959} C_VEL
LIN {X 0,Y 404.403,Z 201.737,A -85,B 0,C 180,E1 -10972.129,E2 -10972.129} C_VEL
LIN {X 0,Y 404.42,Z 201.727,A -85,B 0,C 180,E1 -10974.015,E2 -10974.015} C_VEL
LIN {X 0,Y 404.478,Z 201.72,A -85,B 0,C 180,E1 -10978.009,E2 -10978.009} C_VEL
LIN {X 0,Y 404.607,Z 201.711,A -85,B 0,C 180,E1 -10980,E2 -10980} C_VEL
LIN {X 0,Y 404.414,Z 201.729,A -85,B 0,C 180,E1 -10982.989,E2 -10982.989} C_VEL
LIN {X 0,Y 404.41,Z 201.732,A -85,B 0,C 180,E1 -10986.987,E2 -10986.987} C_VEL
LIN {X 0,Y 404.256,Z 201.752,A -85,B 0,C 180,E1 -10990.012,E2 -10990.012} C_VEL
LIN {X 0,Y 404.265,Z 201.752,A -85,B 0,C 180,E1 -10993.212,E2 -10993.212} C_VEL
LIN {X 0,Y 404.214,Z 201.755,A -85,B 0,C 180,E1 -10997.007,E2 -10997.007} C_VEL
LIN {X 0,Y 404.162,Z 201.758,A -85,B 0,C 180,E1 -11000.352,E2 -11000.352} C_VEL
LIN {X 0,Y 404.168,Z 201.76,A -85,B 0,C 180,E1 -11003.575,E2 -11003.575} C_VEL
LIN {X 0,Y 404.183,Z 201.761,A -85,B 0,C 180,E1 -11005.767,E2 -11005.767} C_VEL
LIN {X 0,Y 404.194,Z 201.745,A -85,B 0,C 180,E1 -11008,E2 -11008} C_VEL
LIN {X 0,Y 404.138,Z 201.768,A -85,B 0,C 180,E1 -11011.558,E2 -11011.558} C_VEL
LIN {X 0,Y 404.185,Z 201.747,A -85,B 0,C 180,E1 -11015.016,E2 -11015.016} C_VEL
LIN {X 0,Y 404.152,Z 201.759,A -85,B 0,C 180,E1 -11018.757,E2 -11018.757} C_VEL
LIN {X 0,Y 404.123,Z 201.77,A -85,B 0,C 180,E1 -11021.6,E2 -11021.6} C_VEL
LIN {X 0,Y 404.145,Z 201.758,A -85,B 0,C 180,E1 -11024.522,E2 -11024.522} C_VEL
LIN {X 0,Y 404.138,Z 201.761,A -85,B 0,C 180,E1 -11027.296,E2 -11027.296} C_VEL
LIN {X 0,Y 404.17,Z 201.765,A -85,B 0,C 180,E1 -11029.956,E2 -11029.956} C_VEL
LIN {X 0,Y 404.139,Z 201.763,A -85,B 0,C 180,E1 -11033.125,E2 -11033.125} C_VEL
LIN {X 0,Y 404.146,Z 201.746,A -85,B 0,C 180,E1 -11036.188,E2 -11036.188} C_VEL
LIN {X 0,Y 404.201,Z 202.023,A -85,B 0,C 180,E1 -11037.017,E2 -11037.017} C_VEL
LIN {X 0,Y 407.279,Z 213.756,A -85,B 0,C 180,E1 -11039.633,E2 -11039.633} C_VEL
LIN {X 0,Y 410.148,Z 225.739,A -85,B 0,C 180,E1 -11042.164,E2 -11042.164} C_VEL
LIN {X 0,Y 411.044,Z 230.041,A -85,B 0,C 180,E1 -11043.035,E2 -11043.035} C_VEL
LIN {X 0,Y 409.77,Z 244.317,A -85,B 0,C 180,E1 -11045.542,E2 -11045.542} C_VEL
LIN {X 0,Y 411.399,Z 252.155,A -85,B 0,C 180,E1 -11045.834,E2 -11045.834} C_VEL
LIN {X 0,Y 415.713,Z 273.707,A -85,B 0,C 180,E1 -11046.502,E2 -11046.502} C_VEL
LIN {X 0,Y 414.041,Z 387.55,A -85,B 0,C 180,E1 -11048.4,E2 -11048.4} C_VEL
LIN {X 0,Y 413.497,Z 401.69,A -85,B 0,C 180,E1 -11048.828,E2 -11048.828} C_VEL
LIN {X 0,Y 412.772,Z 415.769,A -85,B 0,C 180,E1 -11049.464,E2 -11049.464} C_VEL
LIN {X 0,Y 411.863,Z 427.731,A -85,B 0,C 180,E1 -11050.175,E2 -11050.175} C_VEL
LIN {X 0,Y 410.777,Z 440.638,A -85,B 0,C 180,E1 -11051.16,E2 -11051.16} C_VEL
LIN {X 0,Y 409.522,Z 452.334,A -85,B 0,C 180,E1 -11052.265,E2 -11052.265} C_VEL
LIN {X 0,Y 408.401,Z 463.014,A -85,B 0,C 180,E1 -11053.504,E2 -11053.504} C_VEL
LIN {X 0,Y 407.127,Z 473.579,A -85,B 0,C 180,E1 -11054.993,E2 -11054.993} C_VEL
LIN {X 0,Y 406.21,Z 482.307,A -85,B 0,C 180,E1 -11056.493,E2 -11056.493} C_VEL
LIN {X 0,Y 405.117,Z 490.685,A -85,B 0,C 180,E1 -11058.238,E2 -11058.238} C_VEL
LIN {X 0,Y 404.367,Z 497.461,A -85,B 0,C 180,E1 -11059.991,E2 -11059.991} C_VEL
LIN {X 0,Y 404.063,Z 500.337,A -85,B 0,C 180,E1 -11060.87,E2 -11060.87} C_VEL
LIN {X 0,Y 403.176,Z 502.672,A -85,B 0,C 180,E1 -11061.631,E2 -11061.631} C_VEL
LIN {X 0,Y 400.001,Z 506.149,A -85,B 0,C 180,E1 -11062.879,E2 -11062.879} C_VEL
LIN {X 0,Y 397.38,Z 508.484,A -85,B 0,C 180,E1 -11063.907,E2 -11063.907} C_VEL
LIN {X 0,Y 396.217,Z 509.925,A -85,B 0,C 180,E1 -11064.721,E2 -11064.721} C_VEL
LIN {X 0,Y 396.099,Z 510.335,A -85,B 0,C 180,E1 -11065,E2 -11065} C_VEL
LIN {X 0,Y 396.049,Z 512.707,A -85,B 0,C 180,E1 -11066.948,E2 -11066.948} C_VEL
LIN {X 0,Y 395.847,Z 513.961,A -85,B 0,C 180,E1 -11068.982,E2 -11068.982} C_VEL
LIN {X 0,Y 395.846,Z 513.99,A -85,B 0,C 180,E1 -11071.017,E2 -11071.017} C_VEL
LIN {X 0,Y 396.042,Z 512.8,A -85,B 0,C 180,E1 -11073.051,E2 -11073.051} C_VEL
LIN {X 0,Y 396.101,Z 510.369,A -85,B 0,C 180,E1 -11075.089,E2 -11075.089} C_VEL
LIN {X 0,Y 396.511,Z 506.594,A -85,B 0,C 180,E1 -11077.127,E2 -11077.127} C_VEL
LIN {X 0,Y 396.979,Z 501.365,A -85,B 0,C 180,E1 -11079.168,E2 -11079.168} C_VEL
LIN {X 0,Y 397.778,Z 494.501,A -85,B 0,C 180,E1 -11081.206,E2 -11081.206} C_VEL
LIN {X 0,Y 398.712,Z 486.941,A -85,B 0,C 180,E1 -11082.987,E2 -11082.987} C_VEL
LIN {X 0,Y 399.723,Z 478.705,A -85,B 0,C 180,E1 -11084.576,E2 -11084.576} C_VEL
LIN {X 0,Y 400.831,Z 469.613,A -85,B 0,C 180,E1 -11086.03,E2 -11086.03} C_VEL
LIN {X 0,Y 402.144,Z 459.125,A -85,B 0,C 180,E1 -11087.414,E2 -11087.414} C_VEL
LIN {X 0,Y 403.379,Z 447.548,A -85,B 0,C 180,E1 -11088.671,E2 -11088.671} C_VEL
LIN {X 0,Y 404.574,Z 436.229,A -85,B 0,C 180,E1 -11089.667,E2 -11089.667} C_VEL
LIN {X 0,Y 405.642,Z 423.476,A -85,B 0,C 180,E1 -11090.571,E2 -11090.571} C_VEL
LIN {X 0,Y 406.513,Z 410.38,A -85,B 0,C 180,E1 -11091.287,E2 -11091.287} C_VEL
LIN {X 0,Y 407.218,Z 396.226,A -85,B 0,C 180,E1 -11091.847,E2 -11091.847} C_VEL
LIN {X 0,Y 407.651,Z 382.731,A -85,B 0,C 180,E1 -11092.189,E2 -11092.189} C_VEL
LIN {X 0,Y 409.19,Z 273.689,A -85,B 0,C 180,E1 -11094.023,E2 -11094.023} C_VEL
LIN {X 0,Y 403.477,Z 246.244,A -85,B 0,C 180,E1 -11094.917,E2 -11094.917} C_VEL
LIN {X 0,Y 403.152,Z 244.085,A -85,B 0,C 180,E1 -11095.048,E2 -11095.048} C_VEL
LIN {X 0,Y 404.243,Z 231.847,A -85,B 0,C 180,E1 -11097.256,E2 -11097.256} C_VEL
LIN {X 0,Y 401.413,Z 219.141,A -85,B 0,C 180,E1 -11099.932,E2 -11099.932} C_VEL
LIN {X 0,Y 397.96,Z 205.821,A -85,B 0,C 180,E1 -11102.904,E2 -11102.904} C_VEL
LIN {X 0,Y 397.145,Z 202.723,A -85,B 0,C 180,E1 -11103.672,E2 -11103.672} C_VEL
LIN {X 0,Y 397.095,Z 202.643,A -85,B 0,C 180,E1 -11107.209,E2 -11107.209} C_VEL
LIN {X 0,Y 397.099,Z 202.647,A -85,B 0,C 180,E1 -11110.445,E2 -11110.445} C_VEL
LIN {X 0,Y 397.099,Z 202.646,A -85,B 0,C 180,E1 -11113.648,E2 -11113.648} C_VEL
LIN {X 0,Y 397.099,Z 202.638,A -85,B 0,C 180,E1 -11116.52,E2 -11116.52} C_VEL
LIN {X 0,Y 397.109,Z 202.63,A -85,B 0,C 180,E1 -11120.422,E2 -11120.422} C_VEL
LIN {X 0,Y 397.105,Z 202.637,A -85,B 0,C 180,E1 -11124.265,E2 -11124.265} C_VEL
LIN {X 0,Y 397.11,Z 202.635,A -85,B 0,C 180,E1 -11126.726,E2 -11126.726} C_VEL
LIN {X 0,Y 397.128,Z 202.628,A -85,B 0,C 180,E1 -11130.296,E2 -11130.296} C_VEL
LIN {X 0,Y 397.189,Z 202.62,A -85,B 0,C 180,E1 -11132.609,E2 -11132.609} C_VEL
LIN {X 0,Y 397.127,Z 202.636,A -85,B 0,C 180,E1 -11135.981,E2 -11135.981} C_VEL
LIN {X 0,Y 397.132,Z 202.634,A -85,B 0,C 180,E1 -11139.704,E2 -11139.704} C_VEL
LIN {X 0,Y 397.175,Z 202.635,A -85,B 0,C 180,E1 -11142.844,E2 -11142.844} C_VEL
LIN {X 0,Y 397.22,Z 202.632,A -85,B 0,C 180,E1 -11146.679,E2 -11146.679} C_VEL
LIN {X 0,Y 397.211,Z 202.629,A -85,B 0,C 180,E1 -11149.809,E2 -11149.809} C_VEL
LIN {X 0,Y 397.357,Z 202.609,A -85,B 0,C 180,E1 -11152.888,E2 -11152.888} C_VEL
LIN {X 0,Y 397.248,Z 202.626,A -85,B 0,C 180,E1 -11154.925,E2 -11154.925} C_VEL
LIN {X 0,Y 397.445,Z 202.598,A -85,B 0,C 180,E1 -11157.973,E2 -11157.973} C_VEL
LIN {X 0,Y 397.573,Z 202.586,A -85,B 0,C 180,E1 -11160,E2 -11160} C_VEL
LIN {X 0,Y 397.375,Z 202.61,A -85,B 0,C 180,E1 -11163.041,E2 -11163.041} C_VEL
LIN {X 0,Y 397.357,Z 202.611,A -85,B 0,C 180,E1 -11167.112,E2 -11167.112} C_VEL
LIN {X 0,Y 397.211,Z 202.627,A -85,B 0,C 180,E1 -11170.191,E2 -11170.191} C_VEL
LIN {X 0,Y 397.219,Z 202.626,A -85,B 0,C 180,E1 -11173.321,E2 -11173.321} C_VEL
LIN {X 0,Y 397.175,Z 202.631,A -85,B 0,C 180,E1 -11177.155,E2 -11177.155} C_VEL
LIN {X 0,Y 397.096,Z 202.641,A -85,B 0,C 180,E1 -11180.73,E2 -11180.73} C_VEL
LIN {X 0,Y 397.126,Z 202.639,A -85,B 0,C 180,E1 -11184.019,E2 -11184.019} C_VEL
LIN {X 0,Y 397.188,Z 202.614,A -85,B 0,C 180,E1 -11187.39,E2 -11187.39} C_VEL
LIN {X 0,Y 397.072,Z 202.646,A -85,B 0,C 180,E1 -11190.883,E2 -11190.883} C_VEL
LIN {X 0,Y 397.12,Z 202.641,A -85,B 0,C 180,E1 -11194.494,E2 -11194.494} C_VEL
LIN {X 0,Y 397.098,Z 202.636,A -85,B 0,C 180,E1 -11198.275,E2 -11198.275} C_VEL
LIN {X 0,Y 397.083,Z 202.644,A -85,B 0,C 180,E1 -11200.909,E2 -11200.909} C_VEL
LIN {X 0,Y 397.096,Z 202.648,A -85,B 0,C 180,E1 -11203.649,E2 -11203.649} C_VEL
LIN {X 0,Y 397.097,Z 202.643,A -85,B 0,C 180,E1 -11206.522,E2 -11206.522} C_VEL
LIN {X 0,Y 397.107,Z 202.608,A -85,B 0,C 180,E1 -11210.423,E2 -11210.423} C_VEL
LIN {X 0,Y 397.098,Z 202.631,A -85,B 0,C 180,E1 -11214.265,E2 -11214.265} C_VEL
LIN {X 0,Y 397.146,Z 202.931,A -85,B 0,C 180,E1 -11214.541,E2 -11214.541} C_VEL
LIN {X 0,Y 401.09,Z 216.342,A -85,B 0,C 180,E1 -11217.253,E2 -11217.253} C_VEL
LIN {X 0,Y 404.839,Z 230.684,A -85,B 0,C 180,E1 -11219.957,E2 -11219.957} C_VEL
LIN {X 0,Y 405.932,Z 235.424,A -85,B 0,C 180,E1 -11220.809,E2 -11220.809} C_VEL
LIN {X 0,Y 405.017,Z 245.196,A -85,B 0,C 180,E1 -11222.269,E2 -11222.269} C_VEL
LIN {X 0,Y 409.891,Z 274.319,A -85,B 0,C 180,E1 -11223.199,E2 -11223.199} C_VEL
LIN {X 0,Y 407.079,Z 405.226,A -85,B 0,C 180,E1 -11225.658,E2 -11225.658} C_VEL
LIN {X 0,Y 406.381,Z 420.855,A -85,B 0,C 180,E1 -11226.123,E2 -11226.123} C_VEL
LIN {X 0,Y 405.429,Z 435.259,A -85,B 0,C 180,E1 -11226.742,E2 -11226.742} C_VEL
LIN {X 0,Y 404.373,Z 448.945,A -85,B 0,C 180,E1 -11227.521,E2 -11227.521} C_VEL
LIN {X 0,Y 403.082,Z 462.894,A -85,B 0,C 180,E1 -11228.522,E2 -11228.522} C_VEL
LIN {X 0,Y 401.811,Z 475.678,A -85,B 0,C 180,E1 -11229.658,E2 -11229.658} C_VEL
LIN {X 0,Y 400.601,Z 487.53,A -85,B 0,C 180,E1 -11230.929,E2 -11230.929} C_VEL
LIN {X 0,Y 399.496,Z 498.633,A -85,B 0,C 180,E1 -11232.35,E2 -11232.35} C_VEL
LIN {X 0,Y 398.412,Z 508.67,A -85,B 0,C 180,E1 -11233.87,E2 -11233.87} C_VEL
LIN {X 0,Y 397.474,Z 518.581,A -85,B 0,C 180,E1 -11235.668,E2 -11235.668} C_VEL
LIN {X 0,Y 396.855,Z 526.012,A -85,B 0,C 180,E1 -11237.269,E2 -11237.269} C_VEL
LIN {X 0,Y 396.322,Z 533.657,A -85,B 0,C 180,E1 -11239.27,E2 -11239.27} C_VEL
LIN {X 0,Y 395.989,Z 539.911,A -85,B 0,C 180,E1 -11241.324,E2 -11241.324} C_VEL
LIN {X 0,Y 395.885,Z 543.602,A -85,B 0,C 180,E1 -11242.862,E2 -11242.862} C_VEL
LIN {X 0,Y 395.801,Z 547.378,A -85,B 0,C 180,E1 -11244.907,E2 -11244.907} C_VEL
LIN {X 0,Y 395.783,Z 549.865,A -85,B 0,C 180,E1 -11246.947,E2 -11246.947} C_VEL
LIN {X 0,Y 395.875,Z 550.646,A -85,B 0,C 180,E1 -11247.966,E2 -11247.966} C_VEL
LIN {X 0,Y 395.816,Z 551.274,A -85,B 0,C 180,E1 -11250,E2 -11250} C_VEL
LIN {X 0,Y 395.875,Z 550.64,A -85,B 0,C 180,E1 -11252.035,E2 -11252.035} C_VEL
LIN {X 0,Y 395.775,Z 548.765,A -85,B 0,C 180,E1 -11254.073,E2 -11254.073} C_VEL
LIN {X 0,Y 395.896,Z 545.455,A -85,B 0,C 180,E1 -11256.218,E2 -11256.218} C_VEL
LIN {X 0,Y 395.941,Z 541.19,A -85,B 0,C 180,E1 -11258.164,E2 -11258.164} C_VEL
LIN {X 0,Y 396.165,Z 535.3,A -85,B 0,C 180,E1 -11260.219,E2 -11260.219} C_VEL
LIN {X 0,Y 396.769,Z 527.83,A -85,B 0,C 180,E1 -11262.272,E2 -11262.272} C_VEL
LIN {X 0,Y 397.352,Z 519.805,A -85,B 0,C 180,E1 -11264.076,E2 -11264.076} C_VEL
LIN {X 0,Y 398.277,Z 510.145,A -85,B 0,C 180,E1 -11265.874,E2 -11265.874} C_VEL
LIN {X 0,Y 399.272,Z 500.284,A -85,B 0,C 180,E1 -11267.412,E2 -11267.412} C_VEL
LIN {X 0,Y 400.451,Z 488.55,A -85,B 0,C 180,E1 -11268.946,E2 -11268.946} C_VEL
LIN {X 0,Y 401.691,Z 476.904,A -85,B 0,C 180,E1 -11270.215,E2 -11270.215} C_VEL
LIN {X 0,Y 402.954,Z 464.375,A -85,B 0,C 180,E1 -11271.351,E2 -11271.351} C_VEL
LIN {X 0,Y 404.232,Z 450.789,A -85,B 0,C 180,E1 -11272.354,E2 -11272.354} C_VEL
LIN {X 0,Y 405.315,Z 436.776,A -85,B 0,C 180,E1 -11273.177,E2 -11273.177} C_VEL
LIN {X 0,Y 406.273,Z 421.498,A -85,B 0,C 180,E1 -11273.851,E2 -11273.851} C_VEL
LIN {X 0,Y 407.078,Z 406.249,A -85,B 0,C 180,E1 -11274.309,E2 -11274.309} C_VEL
LIN {X 0,Y 409.884,Z 274.359,A -85,B 0,C 180,E1 -11276.789,E2 -11276.789} C_VEL
LIN {X 0,Y 405.007,Z 245.16,A -85,B 0,C 180,E1 -11277.721,E2 -11277.721} C_VEL
LIN {X 0,Y 405.891,Z 235.392,A -85,B 0,C 180,E1 -11279.195,E2 -11279.195} C_VEL
LIN {X 0,Y 402.761,Z 222.47,A -85,B 0,C 180,E1 -11281.566,E2 -11281.566} C_VEL
LIN {X 0,Y 398.74,Z 208.285,A -85,B 0,C 180,E1 -11284.334,E2 -11284.334} C_VEL
LIN {X 0,Y 397.103,Z 202.778,A -85,B 0,C 180,E1 -11285.5,E2 -11285.5} C_VEL
LIN {X 0,Y 397.124,Z 202.613,A -85,B 0,C 180,E1 -11288.86,E2 -11288.86} C_VEL
LIN {X 0,Y 397.067,Z 202.649,A -85,B 0,C 180,E1 -11292.267,E2 -11292.267} C_VEL
LIN {X 0,Y 397.085,Z 202.642,A -85,B 0,C 180,E1 -11295.069,E2 -11295.069} C_VEL
LIN {X 0,Y 397.064,Z 202.638,A -85,B 0,C 180,E1 -11298.021,E2 -11298.021} C_VEL
LIN {X 0,Y 397.13,Z 202.637,A -85,B 0,C 180,E1 -11301.138,E2 -11301.138} C_VEL
LIN {X 0,Y 397.117,Z 202.647,A -85,B 0,C 180,E1 -11304.497,E2 -11304.497} C_VEL
LIN {X 0,Y 397.076,Z 202.63,A -85,B 0,C 180,E1 -11307.928,E2 -11307.928} C_VEL
LIN {X 0,Y 397.12,Z 202.639,A -85,B 0,C 180,E1 -11311.456,E2 -11311.456} C_VEL
LIN {X 0,Y 397.15,Z 202.622,A -85,B 0,C 180,E1 -11314.488,E2 -11314.488} C_VEL
LIN {X 0,Y 397.106,Z 202.643,A -85,B 0,C 180,E1 -11317.086,E2 -11317.086} C_VEL
LIN {X 0,Y 397.146,Z 202.641,A -85,B 0,C 180,E1 -11320.353,E2 -11320.353} C_VEL
LIN {X 0,Y 397.164,Z 202.635,A -85,B 0,C 180,E1 -11323.553,E2 -11323.553} C_VEL
LIN {X 0,Y 397.226,Z 202.625,A -85,B 0,C 180,E1 -11326.703,E2 -11326.703} C_VEL
LIN {X 0,Y 397.215,Z 202.626,A -85,B 0,C 180,E1 -11329.809,E2 -11329.809} C_VEL
LIN {X 0,Y 397.35,Z 202.612,A -85,B 0,C 180,E1 -11332.888,E2 -11332.888} C_VEL
LIN {X 0,Y 397.252,Z 202.618,A -85,B 0,C 180,E1 -11334.925,E2 -11334.925} C_VEL
LIN {X 0,Y 397.447,Z 202.596,A -85,B 0,C 180,E1 -11337.973,E2 -11337.973} C_VEL
LIN {X 0,Y 397.576,Z 202.586,A -85,B 0,C 180,E1 -11340,E2 -11340} C_VEL
LIN {X 0,Y 397.373,Z 202.605,A -85,B 0,C 180,E1 -11343.042,E2 -11343.042} C_VEL
LIN {X 0,Y 397.362,Z 202.609,A -85,B 0,C 180,E1 -11347.112,E2 -11347.112} C_VEL
LIN {X 0,Y 397.216,Z 202.629,A -85,B 0,C 180,E1 -11350.191,E2 -11350.191} C_VEL
LIN {X 0,Y 397.225,Z 202.63,A -85,B 0,C 180,E1 -11353.321,E2 -11353.321} C_VEL
LIN {X 0,Y 397.18,Z 202.633,A -85,B 0,C 180,E1 -11357.155,E2 -11357.155} C_VEL
LIN {X 0,Y 397.107,Z 202.639,A -85,B 0,C 180,E1 -11360.73,E2 -11360.73} C_VEL
LIN {X 0,Y 397.132,Z 202.636,A -85,B 0,C 180,E1 -11364.019,E2 -11364.019} C_VEL
LIN {X 0,Y 397.193,Z 202.62,A -85,B 0,C 180,E1 -11367.39,E2 -11367.39} C_VEL
LIN {X 0,Y 397.078,Z 202.644,A -85,B 0,C 180,E1 -11370.883,E2 -11370.883} C_VEL
LIN {X 0,Y 397.125,Z 202.626,A -85,B 0,C 180,E1 -11374.494,E2 -11374.494} C_VEL
LIN {X 0,Y 397.102,Z 202.645,A -85,B 0,C 180,E1 -11378.275,E2 -11378.275} C_VEL
LIN {X 0,Y 397.088,Z 202.639,A -85,B 0,C 180,E1 -11380.909,E2 -11380.909} C_VEL
LIN {X 0,Y 397.101,Z 202.637,A -85,B 0,C 180,E1 -11383.649,E2 -11383.649} C_VEL
LIN {X 0,Y 397.104,Z 202.644,A -85,B 0,C 180,E1 -11386.521,E2 -11386.521} C_VEL
LIN {X 0,Y 397.115,Z 202.638,A -85,B 0,C 180,E1 -11390.423,E2 -11390.423} C_VEL
LIN {X 0,Y 397.11,Z 202.643,A -85,B 0,C 180,E1 -11394.266,E2 -11394.266} C_VEL
LIN {X 0,Y 397.159,Z 202.787,A -85,B 0,C 180,E1 -11396.476,E2 -11396.476} C_VEL
LIN {X 0,Y 400.412,Z 215.228,A -85,B 0,C 180,E1 -11399.322,E2 -11399.322} C_VEL
LIN {X 0,Y 403.351,Z 227.373,A -85,B 0,C 180,E1 -11401.937,E2 -11401.937} C_VEL
LIN {X 0,Y 404.215,Z 231.384,A -85,B 0,C 180,E1 -11402.766,E2 -11402.766} C_VEL
LIN {X 0,Y 403.308,Z 242.106,A -85,B 0,C 180,E1 -11404.711,E2 -11404.711} C_VEL
LIN {X 0,Y 403.162,Z 244.79,A -85,B 0,C 180,E1 -11405.123,E2 -11405.123} C_VEL
LIN {X 0,Y 408.691,Z 271.445,A -85,B 0,C 180,E1 -11406.002,E2 -11406.002} C_VEL
LIN {X 0,Y 409.27,Z 274.688,A -85,B 0,C 180,E1 -11406.099,E2 -11406.099} C_VEL
LIN {X 0,Y 407.548,Z 387.361,A -85,B 0,C 180,E1 -11408.005,E2 -11408.005} C_VEL
LIN {X 0,Y 406.962,Z 401.646,A -85,B 0,C 180,E1 -11408.437,E2 -11408.437} C_VEL
LIN {X 0,Y 406.204,Z 415.769,A -85,B 0,C 180,E1 -11409.082,E2 -11409.082} C_VEL
LIN {X 0,Y 405.216,Z 428.243,A -85,B 0,C 180,E1 -11409.836,E2 -11409.836} C_VEL
LIN {X 0,Y 404.098,Z 441.097,A -85,B 0,C 180,E1 -11410.836,E2 -11410.836} C_VEL
LIN {X 0,Y 402.782,Z 452.76,A -85,B 0,C 180,E1 -11411.958,E2 -11411.958} C_VEL
LIN {X 0,Y 401.623,Z 463.413,A -85,B 0,C 180,E1 -11413.218,E2 -11413.218} C_VEL
LIN {X 0,Y 400.261,Z 473.963,A -85,B 0,C 180,E1 -11414.729,E2 -11414.729} C_VEL
LIN {X 0,Y 399.304,Z 482.676,A -85,B 0,C 180,E1 -11416.254,E2 -11416.254} C_VEL
LIN {X 0,Y 398.168,Z 491.043,A -85,B 0,C 180,E1 -11418.03,E2 -11418.03} C_VEL
LIN {X 0,Y 397.357,Z 497.812,A -85,B 0,C 180,E1 -11419.812,E2 -11419.812} C_VEL
LIN {X 0,Y 396.734,Z 503.91,A -85,B 0,C 180,E1 -11421.853,E2 -11421.853} C_VEL
LIN {X 0,Y 396.356,Z 508.459,A -85,B 0,C 180,E1 -11423.892,E2 -11423.892} C_VEL
LIN {X 0,Y 396.099,Z 510.335,A -85,B 0,C 180,E1 -11425,E2 -11425} C_VEL
LIN {X 0,Y 395.345,Z 511.534,A -85,B 0,C 180,E1 -11425.834,E2 -11425.834} C_VEL
LIN {X 0,Y 392.379,Z 513.098,A -85,B 0,C 180,E1 -11427.193,E2 -11427.193} C_VEL
LIN {X 0,Y 389.906,Z 513.952,A -85,B 0,C 180,E1 -11428.297,E2 -11428.297} C_VEL
LIN {X 0,Y 388.839,Z 514.332,A -85,B 0,C 180,E1 -11429.156,E2 -11429.156} C_VEL
LIN {X 0,Y 388.749,Z 514.37,A -85,B 0,C 180,E1 -11429.448,E2 -11429.448} C_VEL
LIN {X 0,Y 388.776,Z 514.322,A -85,B 0,C 180,E1 -11431.035,E2 -11431.035} C_VEL
LIN {X 0,Y 388.963,Z 513.133,A -85,B 0,C 180,E1 -11433.107,E2 -11433.107} C_VEL
LIN {X 0,Y 389.048,Z 510.704,A -85,B 0,C 180,E1 -11435.182,E2 -11435.182} C_VEL
LIN {X 0,Y 389.455,Z 506.933,A -85,B 0,C 180,E1 -11437.257,E2 -11437.257} C_VEL
LIN {X 0,Y 389.973,Z 501.708,A -85,B 0,C 180,E1 -11439.334,E2 -11439.334} C_VEL
LIN {X 0,Y 390.805,Z 494.85,A -85,B 0,C 180,E1 -11441.409,E2 -11441.409} C_VEL
LIN {X 0,Y 391.798,Z 487.298,A -85,B 0,C 180,E1 -11443.22,E2 -11443.22} C_VEL
LIN {X 0,Y 392.797,Z 479.487,A -85,B 0,C 180,E1 -11444.763,E2 -11444.763} C_VEL
LIN {X 0,Y 394.002,Z 469.997,A -85,B 0,C 180,E1 -11446.316,E2 -11446.316} C_VEL
LIN {X 0,Y 395.391,Z 459.528,A -85,B 0,C 180,E1 -11447.721,E2 -11447.721} C_VEL
LIN {X 0,Y 396.689,Z 447.976,A -85,B 0,C 180,E1 -11448.998,E2 -11448.998} C_VEL
LIN {X 0,Y 398.07,Z 435.13,A -85,B 0,C 180,E1 -11450.137,E2 -11450.137} C_VEL
LIN {X 0,Y 399.156,Z 422.492,A -85,B 0,C 180,E1 -11451.024,E2 -11451.024} C_VEL
LIN {X 0,Y 400.011,Z 409.698,A -85,B 0,C 180,E1 -11451.718,E2 -11451.718} C_VEL
LIN {X 0,Y 400.732,Z 396.095,A -85,B 0,C 180,E1 -11452.253,E2 -11452.253} C_VEL
LIN {X 0,Y 401.169,Z 382.381,A -85,B 0,C 180,E1 -11452.601,E2 -11452.601} C_VEL
LIN {X 0,Y 402.794,Z 274.93,A -85,B 0,C 180,E1 -11454.434,E2 -11454.434} C_VEL
LIN {X 0,Y 397.73,Z 250.174,A -85,B 0,C 180,E1 -11455.254,E2 -11455.254} C_VEL
LIN {X 0,Y 396.531,Z 244.414,A -85,B 0,C 180,E1 -11455.482,E2 -11455.482} C_VEL
LIN {X 0,Y 397.514,Z 234.03,A -85,B 0,C 180,E1 -11457.365,E2 -11457.365} C_VEL
LIN {X 0,Y 394.957,Z 222.226,A -85,B 0,C 180,E1 -11459.883,E2 -11459.883} C_VEL
LIN {X 0,Y 391.533,Z 208.955,A -85,B 0,C 180,E1 -11462.886,E2 -11462.886} C_VEL
LIN {X 0,Y 390.103,Z 203.638,A -85,B 0,C 180,E1 -11464.176,E2 -11464.176} C_VEL
LIN {X 0,Y 390.043,Z 203.528,A -85,B 0,C 180,E1 -11467.779,E2 -11467.779} C_VEL
LIN {X 0,Y 390.054,Z 203.525,A -85,B 0,C 180,E1 -11470.82,E2 -11470.82} C_VEL
LIN {X 0,Y 390.052,Z 203.526,A -85,B 0,C 180,E1 -11473.885,E2 -11473.885} C_VEL
LIN {X 0,Y 390.054,Z 203.517,A -85,B 0,C 180,E1 -11476.789,E2 -11476.789} C_VEL
LIN {X 0,Y 390.052,Z 203.511,A -85,B 0,C 180,E1 -11479.56,E2 -11479.56} C_VEL
LIN {X 0,Y 390.04,Z 203.525,A -85,B 0,C 180,E1 -11482.448,E2 -11482.448} C_VEL
LIN {X 0,Y 390.063,Z 203.507,A -85,B 0,C 180,E1 -11485.975,E2 -11485.975} C_VEL
LIN {X 0,Y 390.047,Z 203.513,A -85,B 0,C 180,E1 -11489.867,E2 -11489.867} C_VEL
LIN {X 0,Y 390.108,Z 203.509,A -85,B 0,C 180,E1 -11493.231,E2 -11493.231} C_VEL
LIN {X 0,Y 390.101,Z 203.512,A -85,B 0,C 180,E1 -11496.75,E2 -11496.75} C_VEL
LIN {X 0,Y 390.098,Z 203.51,A -85,B 0,C 180,E1 -11499.982,E2 -11499.982} C_VEL
LIN {X 0,Y 390.132,Z 203.507,A -85,B 0,C 180,E1 -11503.248,E2 -11503.248} C_VEL
LIN {X 0,Y 390.188,Z 203.509,A -85,B 0,C 180,E1 -11506.561,E2 -11506.561} C_VEL
LIN {X 0,Y 390.198,Z 203.506,A -85,B 0,C 180,E1 -11510.671,E2 -11510.671} C_VEL
LIN {X 0,Y 390.311,Z 203.486,A -85,B 0,C 180,E1 -11512.759,E2 -11512.759} C_VEL
LIN {X 0,Y 390.22,Z 203.502,A -85,B 0,C 180,E1 -11514.833,E2 -11514.833} C_VEL
LIN {X 0,Y 390.413,Z 203.473,A -85,B 0,C 180,E1 -11517.937,E2 -11517.937} C_VEL
LIN {X 0,Y 390.543,Z 203.462,A -85,B 0,C 180,E1 -11520,E2 -11520} C_VEL
LIN {X 0,Y 390.309,Z 203.49,A -85,B 0,C 180,E1 -11523.096,E2 -11523.096} C_VEL
LIN {X 0,Y 390.323,Z 203.484,A -85,B 0,C 180,E1 -11526.202,E2 -11526.202} C_VEL
LIN {X 0,Y 390.307,Z 203.491,A -85,B 0,C 180,E1 -11528.282,E2 -11528.282} C_VEL
LIN {X 0,Y 390.163,Z 203.507,A -85,B 0,C 180,E1 -11532.483,E2 -11532.483} C_VEL
LIN {X 0,Y 390.132,Z 203.513,A -85,B 0,C 180,E1 -11535.677,E2 -11535.677} C_VEL
LIN {X 0,Y 390.098,Z 203.514,A -85,B 0,C 180,E1 -11538.922,E2 -11538.922} C_VEL
LIN {X 0,Y 390.033,Z 203.525,A -85,B 0,C 180,E1 -11542.234,E2 -11542.234} C_VEL
LIN {X 0,Y 390.112,Z 203.495,A -85,B 0,C 180,E1 -11545.744,E2 -11545.744} C_VEL
LIN {X 0,Y 390.052,Z 203.521,A -85,B 0,C 180,E1 -11549.11,E2 -11549.11} C_VEL
LIN {X 0,Y 390.036,Z 203.504,A -85,B 0,C 180,E1 -11552.722,E2 -11552.722} C_VEL
LIN {X 0,Y 390.05,Z 203.521,A -85,B 0,C 180,E1 -11555.826,E2 -11555.826} C_VEL
LIN {X 0,Y 390.065,Z 203.519,A -85,B 0,C 180,E1 -11559.219,E2 -11559.219} C_VEL
LIN {X 0,Y 390.036,Z 203.514,A -85,B 0,C 180,E1 -11562.375,E2 -11562.375} C_VEL
LIN {X 0,Y 390.039,Z 203.516,A -85,B 0,C 180,E1 -11565.355,E2 -11565.355} C_VEL
LIN {X 0,Y 390.024,Z 203.517,A -85,B 0,C 180,E1 -11568.187,E2 -11568.187} C_VEL
LIN {X 0,Y 390.082,Z 203.486,A -85,B 0,C 180,E1 -11570.908,E2 -11570.908} C_VEL
LIN {X 0,Y 390.081,Z 203.67,A -85,B 0,C 180,E1 -11573.945,E2 -11573.945} C_VEL
LIN {X 0,Y 394.266,Z 217.866,A -85,B 0,C 180,E1 -11576.908,E2 -11576.908} C_VEL
LIN {X 0,Y 397.979,Z 232.03,A -85,B 0,C 180,E1 -11579.639,E2 -11579.639} C_VEL
LIN {X 0,Y 399.209,Z 238.195,A -85,B 0,C 180,E1 -11580.757,E2 -11580.757} C_VEL
LIN {X 0,Y 398.404,Z 245.126,A -85,B 0,C 180,E1 -11581.795,E2 -11581.795} C_VEL
LIN {X 0,Y 402.384,Z 268.468,A -85,B 0,C 180,E1 -11582.573,E2 -11582.573} C_VEL
LIN {X 0,Y 403.485,Z 275.824,A -85,B 0,C 180,E1 -11582.798,E2 -11582.798} C_VEL
LIN {X 0,Y 400.545,Z 405.523,A -85,B 0,C 180,E1 -11585.269,E2 -11585.269} C_VEL
LIN {X 0,Y 399.832,Z 420.969,A -85,B 0,C 180,E1 -11585.741,E2 -11585.741} C_VEL
LIN {X 0,Y 398.777,Z 436.145,A -85,B 0,C 180,E1 -11586.411,E2 -11586.411} C_VEL
LIN {X 0,Y 397.612,Z 450.404,A -85,B 0,C 180,E1 -11587.254,E2 -11587.254} C_VEL
LIN {X 0,Y 396.271,Z 464.01,A -85,B 0,C 180,E1 -11588.271,E2 -11588.271} C_VEL
LIN {X 0,Y 394.968,Z 476.546,A -85,B 0,C 180,E1 -11589.426,E2 -11589.426} C_VEL
LIN {X 0,Y 393.556,Z 489.29,A -85,B 0,C 180,E1 -11590.845,E2 -11590.845} C_VEL
LIN {X 0,Y 392.475,Z 499.955,A -85,B 0,C 180,E1 -11592.278,E2 -11592.278} C_VEL
LIN {X 0,Y 391.342,Z 509.816,A -85,B 0,C 180,E1 -11593.838,E2 -11593.838} C_VEL
LIN {X 0,Y 390.371,Z 519.482,A -85,B 0,C 180,E1 -11595.668,E2 -11595.668} C_VEL
LIN {X 0,Y 389.711,Z 527.509,A -85,B 0,C 180,E1 -11597.503,E2 -11597.503} C_VEL
LIN {X 0,Y 389.288,Z 533.308,A -85,B 0,C 180,E1 -11599.073,E2 -11599.073} C_VEL
LIN {X 0,Y 388.899,Z 539.567,A -85,B 0,C 180,E1 -11601.164,E2 -11601.164} C_VEL
LIN {X 0,Y 388.771,Z 544.369,A -85,B 0,C 180,E1 -11603.252,E2 -11603.252} C_VEL
LIN {X 0,Y 388.703,Z 547.042,A -85,B 0,C 180,E1 -11604.814,E2 -11604.814} C_VEL
LIN {X 0,Y 388.685,Z 549.531,A -85,B 0,C 180,E1 -11606.891,E2 -11606.891} C_VEL
LIN {X 0,Y 388.787,Z 550.313,A -85,B 0,C 180,E1 -11607.929,E2 -11607.929} C_VEL
LIN {X 0,Y 388.744,Z 550.942,A -85,B 0,C 180,E1 -11610,E2 -11610} C_VEL
LIN {X 0,Y 388.787,Z 550.306,A -85,B 0,C 180,E1 -11612.072,E2 -11612.072} C_VEL
LIN {X 0,Y 388.699,Z 548.43,A -85,B 0,C 180,E1 -11614.148,E2 -11614.148} C_VEL
LIN {X 0,Y 388.797,Z 545.304,A -85,B 0,C 180,E1 -11616.227,E2 -11616.227} C_VEL
LIN {X 0,Y 388.874,Z 540.846,A -85,B 0,C 180,E1 -11618.313,E2 -11618.313} C_VEL
LIN {X 0,Y 389.114,Z 534.95,A -85,B 0,C 180,E1 -11620.406,E2 -11620.406} C_VEL
LIN {X 0,Y 389.76,Z 527.471,A -85,B 0,C 180,E1 -11622.497,E2 -11622.497} C_VEL
LIN {X 0,Y 390.372,Z 519.436,A -85,B 0,C 180,E1 -11624.333,E2 -11624.333} C_VEL
LIN {X 0,Y 391.347,Z 509.763,A -85,B 0,C 180,E1 -11626.162,E2 -11626.162} C_VEL
LIN {X 0,Y 392.42,Z 499.887,A -85,B 0,C 180,E1 -11627.726,E2 -11627.726} C_VEL
LIN {X 0,Y 393.64,Z 488.126,A -85,B 0,C 180,E1 -11629.287,E2 -11629.287} C_VEL
LIN {X 0,Y 395.06,Z 475.145,A -85,B 0,C 180,E1 -11630.706,E2 -11630.706} C_VEL
LIN {X 0,Y 396.447,Z 462.291,A -85,B 0,C 180,E1 -11631.856,E2 -11631.856} C_VEL
LIN {X 0,Y 397.813,Z 448.252,A -85,B 0,C 180,E1 -11632.871,E2 -11632.871} C_VEL
LIN {X 0,Y 398.865,Z 434.536,A -85,B 0,C 180,E1 -11633.659,E2 -11633.659} C_VEL
LIN {X 0,Y 399.821,Z 419.791,A -85,B 0,C 180,E1 -11634.295,E2 -11634.295} C_VEL
LIN {X 0,Y 400.561,Z 405.066,A -85,B 0,C 180,E1 -11634.73,E2 -11634.73} C_VEL
LIN {X 0,Y 403.469,Z 275.546,A -85,B 0,C 180,E1 -11637.197,E2 -11637.197} C_VEL
LIN {X 0,Y 398.466,Z 244.956,A -85,B 0,C 180,E1 -11638.203,E2 -11638.203} C_VEL
LIN {X 0,Y 399.216,Z 238.145,A -85,B 0,C 180,E1 -11639.244,E2 -11639.244} C_VEL
LIN {X 0,Y 396.651,Z 226.825,A -85,B 0,C 180,E1 -11641.346,E2 -11641.346} C_VEL
LIN {X 0,Y 392.991,Z 213.578,A -85,B 0,C 180,E1 -11643.949,E2 -11643.949} C_VEL
LIN {X 0,Y 390.049,Z 203.64,A -85,B 0,C 180,E1 -11646.062,E2 -11646.062} C_VEL
LIN {X 0,Y 390.065,Z 203.487,A -85,B 0,C 180,E1 -11649.218,E2 -11649.218} C_VEL
LIN {X 0,Y 390.056,Z 203.522,A -85,B 0,C 180,E1 -11653.21,E2 -11653.21} C_VEL
LIN {X 0,Y 390.055,Z 203.519,A -85,B 0,C 180,E1 -11656.79,E2 -11656.79} C_VEL
LIN {X 0,Y 390.055,Z 203.523,A -85,B 0,C 180,E1 -11659.561,E2 -11659.561} C_VEL
LIN {X 0,Y 390.042,Z 203.512,A -85,B 0,C 180,E1 -11662.449,E2 -11662.449} C_VEL
LIN {X 0,Y 390.066,Z 203.516,A -85,B 0,C 180,E1 -11666.045,E2 -11666.045} C_VEL
LIN {X 0,Y 390.044,Z 203.523,A -85,B 0,C 180,E1 -11669.869,E2 -11669.869} C_VEL
LIN {X 0,Y 390.111,Z 203.491,A -85,B 0,C 180,E1 -11673.232,E2 -11673.232} C_VEL
LIN {X 0,Y 390.104,Z 203.516,A -85,B 0,C 180,E1 -11676.75,E2 -11676.75} C_VEL
LIN {X 0,Y 390.102,Z 203.517,A -85,B 0,C 180,E1 -11679.983,E2 -11679.983} C_VEL
LIN {X 0,Y 390.136,Z 203.509,A -85,B 0,C 180,E1 -11683.248,E2 -11683.248} C_VEL
LIN {X 0,Y 390.192,Z 203.502,A -85,B 0,C 180,E1 -11686.562,E2 -11686.562} C_VEL
LIN {X 0,Y 390.203,Z 203.498,A -85,B 0,C 180,E1 -11690.671,E2 -11690.671} C_VEL
LIN {X 0,Y 390.325,Z 203.484,A -85,B 0,C 180,E1 -11693.798,E2 -11693.798} C_VEL
LIN {X 0,Y 390.416,Z 203.472,A -85,B 0,C 180,E1 -11697.937,E2 -11697.937} C_VEL
LIN {X 0,Y 390.546,Z 203.462,A -85,B 0,C 180,E1 -11700,E2 -11700} C_VEL
LIN {X 0,Y 390.308,Z 203.485,A -85,B 0,C 180,E1 -11703.097,E2 -11703.097} C_VEL
LIN {X 0,Y 390.307,Z 203.485,A -85,B 0,C 180,E1 -11706.642,E2 -11706.642} C_VEL
LIN {X 0,Y 390.203,Z 203.505,A -85,B 0,C 180,E1 -11709.329,E2 -11709.329} C_VEL
LIN {X 0,Y 390.193,Z 203.507,A -85,B 0,C 180,E1 -11713.439,E2 -11713.439} C_VEL
LIN {X 0,Y 390.147,Z 203.511,A -85,B 0,C 180,E1 -11717.308,E2 -11717.308} C_VEL
LIN {X 0,Y 390.087,Z 203.512,A -85,B 0,C 180,E1 -11720.471,E2 -11720.471} C_VEL
LIN {X 0,Y 390.088,Z 203.514,A -85,B 0,C 180,E1 -11723.351,E2 -11723.351} C_VEL
LIN {X 0,Y 390.112,Z 203.51,A -85,B 0,C 180,E1 -11726.768,E2 -11726.768} C_VEL
LIN {X 0,Y 390.038,Z 203.515,A -85,B 0,C 180,E1 -11730.3,E2 -11730.3} C_VEL
LIN {X 0,Y 390.068,Z 203.508,A -85,B 0,C 180,E1 -11734.025,E2 -11734.025} C_VEL
LIN {X 0,Y 390.044,Z 203.524,A -85,B 0,C 180,E1 -11737.551,E2 -11737.551} C_VEL
LIN {X 0,Y 390.056,Z 203.513,A -85,B 0,C 180,E1 -11740.822,E2 -11740.822} C_VEL
LIN {X 0,Y 390.055,Z 203.512,A -85,B 0,C 180,E1 -11743.886,E2 -11743.886} C_VEL
LIN {X 0,Y 390.058,Z 203.518,A -85,B 0,C 180,E1 -11746.79,E2 -11746.79} C_VEL
LIN {X 0,Y 390.057,Z 203.524,A -85,B 0,C 180,E1 -11749.561,E2 -11749.561} C_VEL
LIN {X 0,Y 390.046,Z 203.525,A -85,B 0,C 180,E1 -11752.449,E2 -11752.449} C_VEL
LIN {X 0,Y 390.098,Z 203.667,A -85,B 0,C 180,E1 -11755.947,E2 -11755.947} C_VEL
LIN {X 0,Y 393.578,Z 216.68,A -85,B 0,C 180,E1 -11758.995,E2 -11758.995} C_VEL
LIN {X 0,Y 396.78,Z 230.137,A -85,B 0,C 180,E1 -11761.938,E2 -11761.938} C_VEL
LIN {X 0,Y 397.491,Z 233.441,A -85,B 0,C 180,E1 -11762.632,E2 -11762.632} C_VEL
LIN {X 0,Y 396.519,Z 244.643,A -85,B 0,C 180,E1 -11764.638,E2 -11764.638} C_VEL
LIN {X 0,Y 401.979,Z 271.062,A -85,B 0,C 180,E1 -11765.538,E2 -11765.538} C_VEL
LIN {X 0,Y 402.867,Z 275.985,A -85,B 0,C 180,E1 -11765.69,E2 -11765.69} C_VEL
LIN {X 0,Y 401.06,Z 387.128,A -85,B 0,C 180,E1 -11767.596,E2 -11767.596} C_VEL
LIN {X 0,Y 400.466,Z 401.595,A -85,B 0,C 180,E1 -11768.036,E2 -11768.036} C_VEL
LIN {X 0,Y 399.727,Z 414.937,A -85,B 0,C 180,E1 -11768.642,E2 -11768.642} C_VEL
LIN {X 0,Y 398.719,Z 426.972,A -85,B 0,C 180,E1 -11769.358,E2 -11769.358} C_VEL
LIN {X 0,Y 397.605,Z 440.141,A -85,B 0,C 180,E1 -11770.376,E2 -11770.376} C_VEL
LIN {X 0,Y 396.198,Z 452.026,A -85,B 0,C 180,E1 -11771.514,E2 -11771.514} C_VEL
LIN {X 0,Y 395.121,Z 461.884,A -85,B 0,C 180,E1 -11772.666,E2 -11772.666} C_VEL
LIN {X 0,Y 393.612,Z 472.754,A -85,B 0,C 180,E1 -11774.199,E2 -11774.199} C_VEL
LIN {X 0,Y 392.562,Z 481.727,A -85,B 0,C 180,E1 -11775.749,E2 -11775.749} C_VEL
LIN {X 0,Y 391.342,Z 490.318,A -85,B 0,C 180,E1 -11777.555,E2 -11777.555} C_VEL
LIN {X 0,Y 390.596,Z 496.41,A -85,B 0,C 180,E1 -11779.11,E2 -11779.11} C_VEL
LIN {X 0,Y 389.848,Z 502.882,A -85,B 0,C 180,E1 -11781.185,E2 -11781.185} C_VEL
LIN {X 0,Y 389.427,Z 507.304,A -85,B 0,C 180,E1 -11783.021,E2 -11783.021} C_VEL
LIN {X 0,Y 389.035,Z 510.748,A -85,B 0,C 180,E1 -11784.966,E2 -11784.966} C_VEL
LIN {X 0,Y 388.97,Z 513.041,A -85,B 0,C 180,E1 -11786.892,E2 -11786.892} C_VEL
LIN {X 0,Y 388.777,Z 514.293,A -85,B 0,C 180,E1 -11788.964,E2 -11788.964} C_VEL
LIN {X 0,Y 388.749,Z 514.37,A -85,B 0,C 180,E1 -11789.448,E2 -11789.448} C_VEL
LIN {X 0,Y 388.081,Z 514.466,A -85,B 0,C 180,E1 -11790.313,E2 -11790.313} C_VEL
LIN {X 0,Y 385.273,Z 514.209,A -85,B 0,C 180,E1 -11791.721,E2 -11791.721} C_VEL
LIN {X 0,Y 382.915,Z 513.634,A -85,B 0,C 180,E1 -11792.856,E2 -11792.856} C_VEL
LIN {X 0,Y 381.918,Z 512.912,A -85,B 0,C 180,E1 -11793.729,E2 -11793.729} C_VEL
LIN {X 0,Y 381.844,Z 512.613,A -85,B 0,C 180,E1 -11794.023,E2 -11794.023} C_VEL
LIN {X 0,Y 381.997,Z 511.038,A -85,B 0,C 180,E1 -11795.278,E2 -11795.278} C_VEL
LIN {X 0,Y 382.417,Z 507.271,A -85,B 0,C 180,E1 -11797.391,E2 -11797.391} C_VEL
LIN {X 0,Y 382.949,Z 502.052,A -85,B 0,C 180,E1 -11799.507,E2 -11799.507} C_VEL
LIN {X 0,Y 383.843,Z 495.199,A -85,B 0,C 180,E1 -11801.619,E2 -11801.619} C_VEL
LIN {X 0,Y 384.893,Z 487.654,A -85,B 0,C 180,E1 -11803.462,E2 -11803.462} C_VEL
LIN {X 0,Y 386.069,Z 478.688,A -85,B 0,C 180,E1 -11805.244,E2 -11805.244} C_VEL
LIN {X 0,Y 387.44,Z 468.632,A -85,B 0,C 180,E1 -11806.871,E2 -11806.871} C_VEL
LIN {X 0,Y 388.84,Z 457.83,A -85,B 0,C 180,E1 -11808.302,E2 -11808.302} C_VEL
LIN {X 0,Y 390.347,Z 445.85,A -85,B 0,C 180,E1 -11809.592,E2 -11809.592} C_VEL
LIN {X 0,Y 391.585,Z 434.028,A -85,B 0,C 180,E1 -11810.623,E2 -11810.623} C_VEL
LIN {X 0,Y 392.673,Z 421.689,A -85,B 0,C 180,E1 -11811.48,E2 -11811.48} C_VEL
LIN {X 0,Y 393.642,Z 407.659,A -85,B 0,C 180,E1 -11812.226,E2 -11812.226} C_VEL
LIN {X 0,Y 394.34,Z 394.011,A -85,B 0,C 180,E1 -11812.737,E2 -11812.737} C_VEL
LIN {X 0,Y 394.795,Z 378.433,A -85,B 0,C 180,E1 -11813.09,E2 -11813.09} C_VEL
LIN {X 0,Y 396.423,Z 276.069,A -85,B 0,C 180,E1 -11814.859,E2 -11814.859} C_VEL
LIN {X 0,Y 391.236,Z 250.728,A -85,B 0,C 180,E1 -11815.723,E2 -11815.723} C_VEL
LIN {X 0,Y 389.914,Z 244.333,A -85,B 0,C 180,E1 -11815.986,E2 -11815.986} C_VEL
LIN {X 0,Y 390.699,Z 235.643,A -85,B 0,C 180,E1 -11817.593,E2 -11817.593} C_VEL
LIN {X 0,Y 388.338,Z 224.633,A -85,B 0,C 180,E1 -11819.989,E2 -11819.989} C_VEL
LIN {X 0,Y 385.072,Z 211.943,A -85,B 0,C 180,E1 -11822.907,E2 -11822.907} C_VEL
LIN {X 0,Y 383.072,Z 204.492,A -85,B 0,C 180,E1 -11824.741,E2 -11824.741} C_VEL
LIN {X 0,Y 383.003,Z 204.398,A -85,B 0,C 180,E1 -11828.6,E2 -11828.6} C_VEL
LIN {X 0,Y 382.981,Z 204.401,A -85,B 0,C 180,E1 -11831.347,E2 -11831.347} C_VEL
LIN {X 0,Y 382.993,Z 204.402,A -85,B 0,C 180,E1 -11834.303,E2 -11834.303} C_VEL
LIN {X 0,Y 383.007,Z 204.399,A -85,B 0,C 180,E1 -11837.239,E2 -11837.239} C_VEL
LIN {X 0,Y 383.01,Z 204.385,A -85,B 0,C 180,E1 -11840.413,E2 -11840.413} C_VEL
LIN {X 0,Y 383.022,Z 204.392,A -85,B 0,C 180,E1 -11844.044,E2 -11844.044} C_VEL
LIN {X 0,Y 383.002,Z 204.403,A -85,B 0,C 180,E1 -11847.573,E2 -11847.573} C_VEL
LIN {X 0,Y 383.044,Z 204.373,A -85,B 0,C 180,E1 -11851.507,E2 -11851.507} C_VEL
LIN {X 0,Y 383.046,Z 204.397,A -85,B 0,C 180,E1 -11855.039,E2 -11855.039} C_VEL
LIN {X 0,Y 382.987,Z 204.403,A -85,B 0,C 180,E1 -11858.468,E2 -11858.468} C_VEL
LIN {X 0,Y 383.083,Z 204.39,A -85,B 0,C 180,E1 -11861.827,E2 -11861.827} C_VEL
LIN {X 0,Y 383.105,Z 204.388,A -85,B 0,C 180,E1 -11865.118,E2 -11865.118} C_VEL
LIN {X 0,Y 383.091,Z 204.383,A -85,B 0,C 180,E1 -11868.358,E2 -11868.358} C_VEL
LIN {X 0,Y 383.297,Z 204.36,A -85,B 0,C 180,E1 -11871.933,E2 -11871.933} C_VEL
LIN {X 0,Y 383.192,Z 204.379,A -85,B 0,C 180,E1 -11874.738,E2 -11874.738} C_VEL
LIN {X 0,Y 383.381,Z 204.349,A -85,B 0,C 180,E1 -11877.899,E2 -11877.899} C_VEL
LIN {X 0,Y 383.512,Z 204.338,A -85,B 0,C 180,E1 -11880,E2 -11880} C_VEL
LIN {X 0,Y 383.245,Z 204.369,A -85,B 0,C 180,E1 -11883.153,E2 -11883.153} C_VEL
LIN {X 0,Y 383.28,Z 204.362,A -85,B 0,C 180,E1 -11886.316,E2 -11886.316} C_VEL
LIN {X 0,Y 383.253,Z 204.368,A -85,B 0,C 180,E1 -11888.436,E2 -11888.436} C_VEL
LIN {X 0,Y 383.09,Z 204.389,A -85,B 0,C 180,E1 -11891.642,E2 -11891.642} C_VEL
LIN {X 0,Y 383.103,Z 204.385,A -85,B 0,C 180,E1 -11894.882,E2 -11894.882} C_VEL
LIN {X 0,Y 383.082,Z 204.387,A -85,B 0,C 180,E1 -11898.172,E2 -11898.172} C_VEL
LIN {X 0,Y 382.986,Z 204.398,A -85,B 0,C 180,E1 -11901.531,E2 -11901.531} C_VEL
LIN {X 0,Y 383.045,Z 204.388,A -85,B 0,C 180,E1 -11904.961,E2 -11904.961} C_VEL
LIN {X 0,Y 383.034,Z 204.394,A -85,B 0,C 180,E1 -11908.493,E2 -11908.493} C_VEL
LIN {X 0,Y 383.002,Z 204.38,A -85,B 0,C 180,E1 -11912.15,E2 -11912.15} C_VEL
LIN {X 0,Y 383.012,Z 204.399,A -85,B 0,C 180,E1 -11914.668,E2 -11914.668} C_VEL
LIN {X 0,Y 382.994,Z 204.388,A -85,B 0,C 180,E1 -11917.904,E2 -11917.904} C_VEL
LIN {X 0,Y 382.978,Z 204.394,A -85,B 0,C 180,E1 -11921.348,E2 -11921.348} C_VEL
LIN {X 0,Y 382.99,Z 204.402,A -85,B 0,C 180,E1 -11924.304,E2 -11924.304} C_VEL
LIN {X 0,Y 383.005,Z 204.405,A -85,B 0,C 180,E1 -11927.241,E2 -11927.241} C_VEL
LIN {X 0,Y 383.003,Z 204.363,A -85,B 0,C 180,E1 -11930.416,E2 -11930.416} C_VEL
LIN {X 0,Y 383.046,Z 204.569,A -85,B 0,C 180,E1 -11933.379,E2 -11933.379} C_VEL
LIN {X 0,Y 386.999,Z 217.926,A -85,B 0,C 180,E1 -11936.244,E2 -11936.244} C_VEL
LIN {X 0,Y 390.937,Z 232.635,A -85,B 0,C 180,E1 -11939.165,E2 -11939.165} C_VEL
LIN {X 0,Y 392.458,Z 239.78,A -85,B 0,C 180,E1 -11940.498,E2 -11940.498} C_VEL
LIN {X 0,Y 391.865,Z 244.981,A -85,B 0,C 180,E1 -11941.301,E2 -11941.301} C_VEL
LIN {X 0,Y 395.589,Z 266.848,A -85,B 0,C 180,E1 -11942.059,E2 -11942.059} C_VEL
LIN {X 0,Y 397.095,Z 277.106,A -85,B 0,C 180,E1 -11942.378,E2 -11942.378} C_VEL
LIN {X 0,Y 394.046,Z 405.831,A -85,B 0,C 180,E1 -11944.869,E2 -11944.869} C_VEL
LIN {X 0,Y 393.231,Z 421.942,A -85,B 0,C 180,E1 -11945.377,E2 -11945.377} C_VEL
LIN {X 0,Y 392.141,Z 436.952,A -85,B 0,C 180,E1 -11946.068,E2 -11946.068} C_VEL
LIN {X 0,Y 390.845,Z 451.756,A -85,B 0,C 180,E1 -11946.978,E2 -11946.978} C_VEL
LIN {X 0,Y 389.487,Z 465.081,A -85,B 0,C 180,E1 -11948.012,E2 -11948.012} C_VEL
LIN {X 0,Y 387.977,Z 478.631,A -85,B 0,C 180,E1 -11949.316,E2 -11949.316} C_VEL
LIN {X 0,Y 386.592,Z 490.963,A -85,B 0,C 180,E1 -11950.762,E2 -11950.762} C_VEL
LIN {X 0,Y 385.427,Z 501.373,A -85,B 0,C 180,E1 -11952.217,E2 -11952.217} C_VEL
LIN {X 0,Y 384.135,Z 512.419,A -85,B 0,C 180,E1 -11954.072,E2 -11954.072} C_VEL
LIN {X 0,Y 383.181,Z 521.596,A -85,B 0,C 180,E1 -11955.936,E2 -11955.936} C_VEL
LIN {X 0,Y 382.505,Z 529.226,A -85,B 0,C 180,E1 -11957.802,E2 -11957.802} C_VEL
LIN {X 0,Y 382.074,Z 534.63,A -85,B 0,C 180,E1 -11959.401,E2 -11959.401} C_VEL
LIN {X 0,Y 381.778,Z 540.519,A -85,B 0,C 180,E1 -11961.532,E2 -11961.532} C_VEL
LIN {X 0,Y 381.663,Z 544.98,A -85,B 0,C 180,E1 -11963.657,E2 -11963.657} C_VEL
LIN {X 0,Y 381.614,Z 548.11,A -85,B 0,C 180,E1 -11965.776,E2 -11965.776} C_VEL
LIN {X 0,Y 381.685,Z 549.979,A -85,B 0,C 180,E1 -11967.89,E2 -11967.89} C_VEL
LIN {X 0,Y 381.673,Z 550.61,A -85,B 0,C 180,E1 -11970,E2 -11970} C_VEL
LIN {X 0,Y 381.686,Z 549.973,A -85,B 0,C 180,E1 -11972.111,E2 -11972.111} C_VEL
LIN {X 0,Y 381.624,Z 548.096,A -85,B 0,C 180,E1 -11974.225,E2 -11974.225} C_VEL
LIN {X 0,Y 381.707,Z 544.965,A -85,B 0,C 180,E1 -11976.343,E2 -11976.343} C_VEL
LIN {X 0,Y 381.783,Z 540.501,A -85,B 0,C 180,E1 -11978.469,E2 -11978.469} C_VEL
LIN {X 0,Y 382.075,Z 534.6,A -85,B 0,C 180,E1 -11980.6,E2 -11980.6} C_VEL
LIN {X 0,Y 382.765,Z 527.114,A -85,B 0,C 180,E1 -11982.729,E2 -11982.729} C_VEL
LIN {X 0,Y 383.422,Z 519.069,A -85,B 0,C 180,E1 -11984.598,E2 -11984.598} C_VEL
LIN {X 0,Y 384.442,Z 509.383,A -85,B 0,C 180,E1 -11986.461,E2 -11986.461} C_VEL
LIN {X 0,Y 385.716,Z 498.134,A -85,B 0,C 180,E1 -11988.249,E2 -11988.249} C_VEL
LIN {X 0,Y 387.024,Z 486.624,A -85,B 0,C 180,E1 -11989.768,E2 -11989.768} C_VEL
LIN {X 0,Y 388.369,Z 474.701,A -85,B 0,C 180,E1 -11991.08,E2 -11991.08} C_VEL
LIN {X 0,Y 389.814,Z 461.807,A -85,B 0,C 180,E1 -11992.248,E2 -11992.248} C_VEL
LIN {X 0,Y 391.224,Z 447.708,A -85,B 0,C 180,E1 -11993.279,E2 -11993.279} C_VEL
LIN {X 0,Y 392.409,Z 432.862,A -85,B 0,C 180,E1 -11994.129,E2 -11994.129} C_VEL
LIN {X 0,Y 393.431,Z 418.093,A -85,B 0,C 180,E1 -11994.751,E2 -11994.751} C_VEL
LIN {X 0,Y 394.118,Z 402.443,A -85,B 0,C 180,E1 -11995.198,E2 -11995.198} C_VEL
LIN {X 0,Y 397.042,Z 277.353,A -85,B 0,C 180,E1 -11997.607,E2 -11997.607} C_VEL
LIN {X 0,Y 392.95,Z 251.015,A -85,B 0,C 180,E1 -11998.451,E2 -11998.451} C_VEL
LIN {X 0,Y 391.929,Z 244.945,A -85,B 0,C 180,E1 -11998.686,E2 -11998.686} C_VEL
LIN {X 0,Y 392.468,Z 239.711,A -85,B 0,C 180,E1 -11999.502,E2 -11999.502} C_VEL
LIN {X 0,Y 389.833,Z 228.29,A -85,B 0,C 180,E1 -12001.672,E2 -12001.672} C_VEL
LIN {X 0,Y 386.148,Z 215.022,A -85,B 0,C 180,E1 -12004.347,E2 -12004.347} C_VEL
LIN {X 0,Y 383.02,Z 204.505,A -85,B 0,C 180,E1 -12006.646,E2 -12006.646} C_VEL
LIN {X 0,Y 382.994,Z 204.364,A -85,B 0,C 180,E1 -12009.96,E2 -12009.96} C_VEL
LIN {X 0,Y 383.004,Z 204.406,A -85,B 0,C 180,E1 -12012.779,E2 -12012.779} C_VEL
LIN {X 0,Y 382.995,Z 204.402,A -85,B 0,C 180,E1 -12015.789,E2 -12015.789} C_VEL
LIN {X 0,Y 382.986,Z 204.396,A -85,B 0,C 180,E1 -12018.796,E2 -12018.796} C_VEL
LIN {X 0,Y 382.998,Z 204.389,A -85,B 0,C 180,E1 -12022.096,E2 -12022.096} C_VEL
LIN {X 0,Y 383.016,Z 204.4,A -85,B 0,C 180,E1 -12025.332,E2 -12025.332} C_VEL
LIN {X 0,Y 382.981,Z 204.401,A -85,B 0,C 180,E1 -12029.081,E2 -12029.081} C_VEL
LIN {X 0,Y 383.054,Z 204.372,A -85,B 0,C 180,E1 -12032.698,E2 -12032.698} C_VEL
LIN {X 0,Y 383.049,Z 204.387,A -85,B 0,C 180,E1 -12035.04,E2 -12035.04} C_VEL
LIN {X 0,Y 382.991,Z 204.398,A -85,B 0,C 180,E1 -12038.469,E2 -12038.469} C_VEL
LIN {X 0,Y 383.087,Z 204.387,A -85,B 0,C 180,E1 -12041.828,E2 -12041.828} C_VEL
LIN {X 0,Y 383.108,Z 204.385,A -85,B 0,C 180,E1 -12045.118,E2 -12045.118} C_VEL
LIN {X 0,Y 383.095,Z 204.389,A -85,B 0,C 180,E1 -12048.358,E2 -12048.358} C_VEL
LIN {X 0,Y 383.262,Z 204.372,A -85,B 0,C 180,E1 -12051.976,E2 -12051.976} C_VEL
LIN {X 0,Y 383.196,Z 204.368,A -85,B 0,C 180,E1 -12054.739,E2 -12054.739} C_VEL
LIN {X 0,Y 383.383,Z 204.348,A -85,B 0,C 180,E1 -12057.899,E2 -12057.899} C_VEL
LIN {X 0,Y 383.515,Z 204.337,A -85,B 0,C 180,E1 -12060,E2 -12060} C_VEL
LIN {X 0,Y 383.245,Z 204.364,A -85,B 0,C 180,E1 -12063.154,E2 -12063.154} C_VEL
LIN {X 0,Y 383.267,Z 204.362,A -85,B 0,C 180,E1 -12066.637,E2 -12066.637} C_VEL
LIN {X 0,Y 383.258,Z 204.364,A -85,B 0,C 180,E1 -12068.436,E2 -12068.436} C_VEL
LIN {X 0,Y 383.095,Z 204.383,A -85,B 0,C 180,E1 -12071.642,E2 -12071.642} C_VEL
LIN {X 0,Y 383.109,Z 204.389,A -85,B 0,C 180,E1 -12074.882,E2 -12074.882} C_VEL
LIN {X 0,Y 383.061,Z 204.392,A -85,B 0,C 180,E1 -12078.174,E2 -12078.174} C_VEL
LIN {X 0,Y 382.998,Z 204.403,A -85,B 0,C 180,E1 -12081.531,E2 -12081.531} C_VEL
LIN {X 0,Y 383.051,Z 204.396,A -85,B 0,C 180,E1 -12084.961,E2 -12084.961} C_VEL
LIN {X 0,Y 383.028,Z 204.377,A -85,B 0,C 180,E1 -12088.27,E2 -12088.27} C_VEL
LIN {X 0,Y 383.009,Z 204.401,A -85,B 0,C 180,E1 -12092.15,E2 -12092.15} C_VEL
LIN {X 0,Y 383.018,Z 204.381,A -85,B 0,C 180,E1 -12094.668,E2 -12094.668} C_VEL
LIN {X 0,Y 383,Z 204.401,A -85,B 0,C 180,E1 -12097.904,E2 -12097.904} C_VEL
LIN {X 0,Y 382.984,Z 204.403,A -85,B 0,C 180,E1 -12101.348,E2 -12101.348} C_VEL
LIN {X 0,Y 382.996,Z 204.391,A -85,B 0,C 180,E1 -12104.304,E2 -12104.304} C_VEL
LIN {X 0,Y 383.011,Z 204.392,A -85,B 0,C 180,E1 -12107.24,E2 -12107.24} C_VEL
LIN {X 0,Y 383.016,Z 204.394,A -85,B 0,C 180,E1 -12110.414,E2 -12110.414} C_VEL
LIN {X 0,Y 383.027,Z 204.394,A -85,B 0,C 180,E1 -12114.045,E2 -12114.045} C_VEL
LIN {X 0,Y 383.096,Z 204.593,A -85,B 0,C 180,E1 -12115.418,E2 -12115.418} C_VEL
LIN {X 0,Y 386.749,Z 218.146,A -85,B 0,C 180,E1 -12118.659,E2 -12118.659} C_VEL
LIN {X 0,Y 389.712,Z 230.647,A -85,B 0,C 180,E1 -12121.452,E2 -12121.452} C_VEL
LIN {X 0,Y 390.686,Z 235.075,A -85,B 0,C 180,E1 -12122.405,E2 -12122.405} C_VEL
LIN {X 0,Y 389.887,Z 244.401,A -85,B 0,C 180,E1 -12124.122,E2 -12124.122} C_VEL
LIN {X 0,Y 395.311,Z 270.357,A -85,B 0,C 180,E1 -12125.054,E2 -12125.054} C_VEL
LIN {X 0,Y 396.477,Z 277.07,A -85,B 0,C 180,E1 -12125.264,E2 -12125.264} C_VEL
LIN {X 0,Y 394.553,Z 388.185,A -85,B 0,C 180,E1 -12127.206,E2 -12127.206} C_VEL
LIN {X 0,Y 393.921,Z 402.313,A -85,B 0,C 180,E1 -12127.651,E2 -12127.651} C_VEL
LIN {X 0,Y 393.13,Z 415.802,A -85,B 0,C 180,E1 -12128.283,E2 -12128.283} C_VEL
LIN {X 0,Y 391.967,Z 429.257,A -85,B 0,C 180,E1 -12129.123,E2 -12129.123} C_VEL
LIN {X 0,Y 390.779,Z 442.009,A -85,B 0,C 180,E1 -12130.156,E2 -12130.156} C_VEL
LIN {X 0,Y 389.336,Z 453.604,A -85,B 0,C 180,E1 -12131.312,E2 -12131.312} C_VEL
LIN {X 0,Y 388.067,Z 464.209,A -85,B 0,C 180,E1 -12132.613,E2 -12132.613} C_VEL
LIN {X 0,Y 386.588,Z 474.722,A -85,B 0,C 180,E1 -12134.175,E2 -12134.175} C_VEL
LIN {X 0,Y 385.498,Z 483.41,A -85,B 0,C 180,E1 -12135.752,E2 -12135.752} C_VEL
LIN {X 0,Y 384.263,Z 491.756,A -85,B 0,C 180,E1 -12137.59,E2 -12137.59} C_VEL
LIN {X 0,Y 383.386,Z 498.509,A -85,B 0,C 180,E1 -12139.437,E2 -12139.437} C_VEL
LIN {X 0,Y 382.687,Z 504.596,A -85,B 0,C 180,E1 -12141.551,E2 -12141.551} C_VEL
LIN {X 0,Y 382.24,Z 509.137,A -85,B 0,C 180,E1 -12143.666,E2 -12143.666} C_VEL
LIN {X 0,Y 381.869,Z 512.292,A -85,B 0,C 180,E1 -12145.778,E2 -12145.778} C_VEL
LIN {X 0,Y 381.813,Z 514.152,A -85,B 0,C 180,E1 -12147.89,E2 -12147.89} C_VEL
LIN {X 0,Y 381.68,Z 514.791,A -85,B 0,C 180,E1 -12150,E2 -12150} C_VEL
LIN {X 0,Y 381.805,Z 514.212,A -85,B 0,C 180,E1 -12152.109,E2 -12152.109} C_VEL
LIN {X 0,Y 381.844,Z 512.613,A -85,B 0,C 180,E1 -12154.023,E2 -12154.023} C_VEL
LIN {X 0,Y 381.232,Z 511.646,A -85,B 0,C 180,E1 -12154.894,E2 -12154.894} C_VEL
LIN {X 0,Y 378.569,Z 509.654,A -85,B 0,C 180,E1 -12156.305,E2 -12156.305} C_VEL
LIN {X 0,Y 376.391,Z 507.722,A -85,B 0,C 180,E1 -12157.431,E2 -12157.431} C_VEL
LIN {X 0,Y 375.57,Z 505.933,A -85,B 0,C 180,E1 -12158.287,E2 -12158.287} C_VEL
LIN {X 0,Y 375.564,Z 505.277,A -85,B 0,C 180,E1 -12158.573,E2 -12158.573} C_VEL
LIN {X 0,Y 376.36,Z 499.189,A -85,B 0,C 180,E1 -12160.762,E2 -12160.762} C_VEL
LIN {X 0,Y 377.278,Z 492.521,A -85,B 0,C 180,E1 -12162.643,E2 -12162.643} C_VEL
LIN {X 0,Y 378.555,Z 484.266,A -85,B 0,C 180,E1 -12164.514,E2 -12164.514} C_VEL
LIN {X 0,Y 379.692,Z 475.691,A -85,B 0,C 180,E1 -12166.119,E2 -12166.119} C_VEL
LIN {X 0,Y 381.237,Z 465.309,A -85,B 0,C 180,E1 -12167.708,E2 -12167.708} C_VEL
LIN {X 0,Y 382.583,Z 454.866,A -85,B 0,C 180,E1 -12169.029,E2 -12169.029} C_VEL
LIN {X 0,Y 384.003,Z 443.503,A -85,B 0,C 180,E1 -12170.208,E2 -12170.208} C_VEL
LIN {X 0,Y 385.282,Z 431.058,A -85,B 0,C 180,E1 -12171.256,E2 -12171.256} C_VEL
LIN {X 0,Y 386.498,Z 417.105,A -85,B 0,C 180,E1 -12172.167,E2 -12172.167} C_VEL
LIN {X 0,Y 387.383,Z 403.73,A -85,B 0,C 180,E1 -12172.816,E2 -12172.816} C_VEL
LIN {X 0,Y 388.042,Z 390.258,A -85,B 0,C 180,E1 -12173.269,E2 -12173.269} C_VEL
LIN {X 0,Y 388.547,Z 368.409,A -85,B 0,C 180,E1 -12173.696,E2 -12173.696} C_VEL
LIN {X 0,Y 390.077,Z 277.166,A -85,B 0,C 180,E1 -12175.3,E2 -12175.3} C_VEL
LIN {X 0,Y 384.166,Z 248.514,A -85,B 0,C 180,E1 -12176.309,E2 -12176.309} C_VEL
LIN {X 0,Y 383.357,Z 244.304,A -85,B 0,C 180,E1 -12176.5,E2 -12176.5} C_VEL
LIN {X 0,Y 383.945,Z 237.468,A -85,B 0,C 180,E1 -12177.789,E2 -12177.789} C_VEL
LIN {X 0,Y 381.716,Z 227.131,A -85,B 0,C 180,E1 -12180.078,E2 -12180.078} C_VEL
LIN {X 0,Y 378.563,Z 214.732,A -85,B 0,C 180,E1 -12182.976,E2 -12182.976} C_VEL
LIN {X 0,Y 376.029,Z 205.399,A -85,B 0,C 180,E1 -12185.305,E2 -12185.305} C_VEL
LIN {X 0,Y 375.973,Z 205.277,A -85,B 0,C 180,E1 -12188.27,E2 -12188.27} C_VEL
LIN {X 0,Y 375.931,Z 205.276,A -85,B 0,C 180,E1 -12191.6,E2 -12191.6} C_VEL
LIN {X 0,Y 375.924,Z 205.274,A -85,B 0,C 180,E1 -12195.268,E2 -12195.268} C_VEL
LIN {X 0,Y 375.931,Z 205.283,A -85,B 0,C 180,E1 -12198.398,E2 -12198.398} C_VEL
LIN {X 0,Y 375.97,Z 205.275,A -85,B 0,C 180,E1 -12201.729,E2 -12201.729} C_VEL
LIN {X 0,Y 375.975,Z 205.258,A -85,B 0,C 180,E1 -12205.332,E2 -12205.332} C_VEL
LIN {X 0,Y 375.955,Z 205.279,A -85,B 0,C 180,E1 -12208.438,E2 -12208.438} C_VEL
LIN {X 0,Y 375.997,Z 205.254,A -85,B 0,C 180,E1 -12212.141,E2 -12212.141} C_VEL
LIN {X 0,Y 376.001,Z 205.273,A -85,B 0,C 180,E1 -12214.538,E2 -12214.538} C_VEL
LIN {X 0,Y 375.957,Z 205.277,A -85,B 0,C 180,E1 -12218.045,E2 -12218.045} C_VEL
LIN {X 0,Y 376.018,Z 205.271,A -85,B 0,C 180,E1 -12221.473,E2 -12221.473} C_VEL
LIN {X 0,Y 376.053,Z 205.263,A -85,B 0,C 180,E1 -12224.832,E2 -12224.832} C_VEL
LIN {X 0,Y 376.043,Z 205.261,A -85,B 0,C 180,E1 -12228.136,E2 -12228.136} C_VEL
LIN {X 0,Y 376.251,Z 205.238,A -85,B 0,C 180,E1 -12231.877,E2 -12231.877} C_VEL
LIN {X 0,Y 376.165,Z 205.255,A -85,B 0,C 180,E1 -12234.64,E2 -12234.64} C_VEL
LIN {X 0,Y 376.347,Z 205.225,A -85,B 0,C 180,E1 -12237.859,E2 -12237.859} C_VEL
LIN {X 0,Y 376.482,Z 205.213,A -85,B 0,C 180,E1 -12240,E2 -12240} C_VEL
LIN {X 0,Y 376.183,Z 205.249,A -85,B 0,C 180,E1 -12243.213,E2 -12243.213} C_VEL
LIN {X 0,Y 376.24,Z 205.24,A -85,B 0,C 180,E1 -12246.435,E2 -12246.435} C_VEL
LIN {X 0,Y 376.198,Z 205.245,A -85,B 0,C 180,E1 -12248.595,E2 -12248.595} C_VEL
LIN {X 0,Y 376.043,Z 205.269,A -85,B 0,C 180,E1 -12251.863,E2 -12251.863} C_VEL
LIN {X 0,Y 376.051,Z 205.264,A -85,B 0,C 180,E1 -12255.168,E2 -12255.168} C_VEL
LIN {X 0,Y 376.017,Z 205.27,A -85,B 0,C 180,E1 -12258.526,E2 -12258.526} C_VEL
LIN {X 0,Y 375.956,Z 205.275,A -85,B 0,C 180,E1 -12261.955,E2 -12261.955} C_VEL
LIN {X 0,Y 375.999,Z 205.255,A -85,B 0,C 180,E1 -12265.461,E2 -12265.461} C_VEL
LIN {X 0,Y 375.964,Z 205.276,A -85,B 0,C 180,E1 -12269.079,E2 -12269.079} C_VEL
LIN {X 0,Y 375.943,Z 205.259,A -85,B 0,C 180,E1 -12272.829,E2 -12272.829} C_VEL
LIN {X 0,Y 375.951,Z 205.282,A -85,B 0,C 180,E1 -12275.416,E2 -12275.416} C_VEL
LIN {X 0,Y 375.969,Z 205.265,A -85,B 0,C 180,E1 -12278.271,E2 -12278.271} C_VEL
LIN {X 0,Y 375.929,Z 205.27,A -85,B 0,C 180,E1 -12281.601,E2 -12281.601} C_VEL
LIN {X 0,Y 375.921,Z 205.274,A -85,B 0,C 180,E1 -12285.269,E2 -12285.269} C_VEL
LIN {X 0,Y 375.92,Z 205.265,A -85,B 0,C 180,E1 -12288.401,E2 -12288.401} C_VEL
LIN {X 0,Y 375.957,Z 205.262,A -85,B 0,C 180,E1 -12291.912,E2 -12291.912} C_VEL
LIN {X 0,Y 375.97,Z 205.46,A -85,B 0,C 180,E1 -12292.777,E2 -12292.777} C_VEL
LIN {X 0,Y 379.611,Z 217.621,A -85,B 0,C 180,E1 -12295.472,E2 -12295.472} C_VEL
LIN {X 0,Y 382.76,Z 229.005,A -85,B 0,C 180,E1 -12297.828,E2 -12297.828} C_VEL
LIN {X 0,Y 385.371,Z 239.574,A -85,B 0,C 180,E1 -12299.901,E2 -12299.901} C_VEL
LIN {X 0,Y 385.692,Z 241.336,A -85,B 0,C 180,E1 -12300.229,E2 -12300.229} C_VEL
LIN {X 0,Y 385.378,Z 245.041,A -85,B 0,C 180,E1 -12300.808,E2 -12300.808} C_VEL
LIN {X 0,Y 389.408,Z 269.113,A -85,B 0,C 180,E1 -12301.652,E2 -12301.652} C_VEL
LIN {X 0,Y 390.723,Z 277.646,A -85,B 0,C 180,E1 -12301.929,E2 -12301.929} C_VEL
LIN {X 0,Y 387.563,Z 406.137,A -85,B 0,C 180,E1 -12304.454,E2 -12304.454} C_VEL
LIN {X 0,Y 386.711,Z 422.02,A -85,B 0,C 180,E1 -12304.97,E2 -12304.97} C_VEL
LIN {X 0,Y 385.669,Z 435.987,A -85,B 0,C 180,E1 -12305.618,E2 -12305.618} C_VEL
LIN {X 0,Y 384.273,Z 451.258,A -85,B 0,C 180,E1 -12306.561,E2 -12306.561} C_VEL
LIN {X 0,Y 382.833,Z 464.626,A -85,B 0,C 180,E1 -12307.61,E2 -12307.61} C_VEL
LIN {X 0,Y 381.259,Z 478.211,A -85,B 0,C 180,E1 -12308.934,E2 -12308.934} C_VEL
LIN {X 0,Y 379.874,Z 489.553,A -85,B 0,C 180,E1 -12310.267,E2 -12310.267} C_VEL
LIN {X 0,Y 378.594,Z 500.989,A -85,B 0,C 180,E1 -12311.885,E2 -12311.885} C_VEL
LIN {X 0,Y 377.216,Z 512.051,A -85,B 0,C 180,E1 -12313.772,E2 -12313.772} C_VEL
LIN {X 0,Y 376.205,Z 521.238,A -85,B 0,C 180,E1 -12315.669,E2 -12315.669} C_VEL
LIN {X 0,Y 375.498,Z 528.874,A -85,B 0,C 180,E1 -12317.571,E2 -12317.571} C_VEL
LIN {X 0,Y 374.895,Z 535.935,A -85,B 0,C 180,E1 -12319.742,E2 -12319.742} C_VEL
LIN {X 0,Y 374.658,Z 541.462,A -85,B 0,C 180,E1 -12321.913,E2 -12321.913} C_VEL
LIN {X 0,Y 374.57,Z 545.354,A -85,B 0,C 180,E1 -12323.949,E2 -12323.949} C_VEL
LIN {X 0,Y 374.539,Z 547.776,A -85,B 0,C 180,E1 -12325.696,E2 -12325.696} C_VEL
LIN {X 0,Y 374.584,Z 549.646,A -85,B 0,C 180,E1 -12327.85,E2 -12327.85} C_VEL
LIN {X 0,Y 374.605,Z 550.279,A -85,B 0,C 180,E1 -12330,E2 -12330} C_VEL
LIN {X 0,Y 374.585,Z 549.639,A -85,B 0,C 180,E1 -12332.151,E2 -12332.151} C_VEL
LIN {X 0,Y 374.55,Z 547.761,A -85,B 0,C 180,E1 -12334.305,E2 -12334.305} C_VEL
LIN {X 0,Y 374.623,Z 544.626,A -85,B 0,C 180,E1 -12336.463,E2 -12336.463} C_VEL
LIN {X 0,Y 374.711,Z 540.158,A -85,B 0,C 180,E1 -12338.63,E2 -12338.63} C_VEL
LIN {X 0,Y 375.048,Z 534.251,A -85,B 0,C 180,E1 -12340.801,E2 -12340.801} C_VEL
LIN {X 0,Y 375.731,Z 526.756,A -85,B 0,C 180,E1 -12342.971,E2 -12342.971} C_VEL
LIN {X 0,Y 376.474,Z 518.703,A -85,B 0,C 180,E1 -12344.874,E2 -12344.874} C_VEL
LIN {X 0,Y 377.538,Z 509.004,A -85,B 0,C 180,E1 -12346.771,E2 -12346.771} C_VEL
LIN {X 0,Y 378.859,Z 497.959,A -85,B 0,C 180,E1 -12348.558,E2 -12348.558} C_VEL
LIN {X 0,Y 380.209,Z 486.207,A -85,B 0,C 180,E1 -12350.138,E2 -12350.138} C_VEL
LIN {X 0,Y 381.67,Z 474.259,A -85,B 0,C 180,E1 -12351.468,E2 -12351.468} C_VEL
LIN {X 0,Y 383.198,Z 461.326,A -85,B 0,C 180,E1 -12352.653,E2 -12352.653} C_VEL
LIN {X 0,Y 384.667,Z 447.168,A -85,B 0,C 180,E1 -12353.7,E2 -12353.7} C_VEL
LIN {X 0,Y 385.865,Z 432.654,A -85,B 0,C 180,E1 -12354.542,E2 -12354.542} C_VEL
LIN {X 0,Y 386.954,Z 417.291,A -85,B 0,C 180,E1 -12355.194,E2 -12355.194} C_VEL
LIN {X 0,Y 387.643,Z 402.722,A -85,B 0,C 180,E1 -12355.613,E2 -12355.613} C_VEL
LIN {X 0,Y 390.667,Z 277.815,A -85,B 0,C 180,E1 -12358.057,E2 -12358.057} C_VEL
LIN {X 0,Y 385.758,Z 247.316,A -85,B 0,C 180,E1 -12359.075,E2 -12359.075} C_VEL
LIN {X 0,Y 385.414,Z 244.682,A -85,B 0,C 180,E1 -12359.218,E2 -12359.218} C_VEL
LIN {X 0,Y 385.668,Z 241.26,A -85,B 0,C 180,E1 -12359.774,E2 -12359.774} C_VEL
LIN {X 0,Y 383.225,Z 230.725,A -85,B 0,C 180,E1 -12361.819,E2 -12361.819} C_VEL
LIN {X 0,Y 379.144,Z 215.837,A -85,B 0,C 180,E1 -12364.892,E2 -12364.892} C_VEL
LIN {X 0,Y 375.966,Z 205.379,A -85,B 0,C 180,E1 -12367.256,E2 -12367.256} C_VEL
LIN {X 0,Y 375.926,Z 205.25,A -85,B 0,C 180,E1 -12370.869,E2 -12370.869} C_VEL
LIN {X 0,Y 375.928,Z 205.276,A -85,B 0,C 180,E1 -12373.766,E2 -12373.766} C_VEL
LIN {X 0,Y 375.933,Z 205.278,A -85,B 0,C 180,E1 -12376.811,E2 -12376.811} C_VEL
LIN {X 0,Y 375.961,Z 205.28,A -85,B 0,C 180,E1 -12380.538,E2 -12380.538} C_VEL
LIN {X 0,Y 375.962,Z 205.274,A -85,B 0,C 180,E1 -12383.496,E2 -12383.496} C_VEL
LIN {X 0,Y 375.958,Z 205.275,A -85,B 0,C 180,E1 -12385.889,E2 -12385.889} C_VEL
LIN {X 0,Y 375.963,Z 205.276,A -85,B 0,C 180,E1 -12389.687,E2 -12389.687} C_VEL
LIN {X 0,Y 375.994,Z 205.258,A -85,B 0,C 180,E1 -12392.141,E2 -12392.141} C_VEL
LIN {X 0,Y 376.003,Z 205.254,A -85,B 0,C 180,E1 -12394.539,E2 -12394.539} C_VEL
LIN {X 0,Y 375.961,Z 205.275,A -85,B 0,C 180,E1 -12398.046,E2 -12398.046} C_VEL
LIN {X 0,Y 376.022,Z 205.269,A -85,B 0,C 180,E1 -12401.474,E2 -12401.474} C_VEL
LIN {X 0,Y 376.056,Z 205.264,A -85,B 0,C 180,E1 -12404.833,E2 -12404.833} C_VEL
LIN {X 0,Y 376.048,Z 205.269,A -85,B 0,C 180,E1 -12408.137,E2 -12408.137} C_VEL
LIN {X 0,Y 376.217,Z 205.248,A -85,B 0,C 180,E1 -12411.919,E2 -12411.919} C_VEL
LIN {X 0,Y 376.168,Z 205.244,A -85,B 0,C 180,E1 -12414.64,E2 -12414.64} C_VEL
LIN {X 0,Y 376.349,Z 205.225,A -85,B 0,C 180,E1 -12417.86,E2 -12417.86} C_VEL
LIN {X 0,Y 376.485,Z 205.212,A -85,B 0,C 180,E1 -12420,E2 -12420} C_VEL
LIN {X 0,Y 376.183,Z 205.243,A -85,B 0,C 180,E1 -12423.213,E2 -12423.213} C_VEL
LIN {X 0,Y 376.232,Z 205.239,A -85,B 0,C 180,E1 -12426.628,E2 -12426.628} C_VEL
LIN {X 0,Y 376.204,Z 205.243,A -85,B 0,C 180,E1 -12428.595,E2 -12428.595} C_VEL
LIN {X 0,Y 376.048,Z 205.26,A -85,B 0,C 180,E1 -12431.864,E2 -12431.864} C_VEL
LIN {X 0,Y 376.057,Z 205.263,A -85,B 0,C 180,E1 -12435.168,E2 -12435.168} C_VEL
LIN {X 0,Y 376.007,Z 205.272,A -85,B 0,C 180,E1 -12438.527,E2 -12438.527} C_VEL
LIN {X 0,Y 375.967,Z 205.277,A -85,B 0,C 180,E1 -12441.954,E2 -12441.954} C_VEL
LIN {X 0,Y 376.005,Z 205.273,A -85,B 0,C 180,E1 -12445.461,E2 -12445.461} C_VEL
LIN {X 0,Y 375.96,Z 205.255,A -85,B 0,C 180,E1 -12449.08,E2 -12449.08} C_VEL
LIN {X 0,Y 375.949,Z 205.277,A -85,B 0,C 180,E1 -12452.829,E2 -12452.829} C_VEL
LIN {X 0,Y 375.958,Z 205.262,A -85,B 0,C 180,E1 -12455.416,E2 -12455.416} C_VEL
LIN {X 0,Y 375.974,Z 205.275,A -85,B 0,C 180,E1 -12458.271,E2 -12458.271} C_VEL
LIN {X 0,Y 375.935,Z 205.281,A -85,B 0,C 180,E1 -12461.601,E2 -12461.601} C_VEL
LIN {X 0,Y 375.927,Z 205.279,A -85,B 0,C 180,E1 -12465.269,E2 -12465.269} C_VEL
LIN {X 0,Y 375.935,Z 205.274,A -85,B 0,C 180,E1 -12468.4,E2 -12468.4} C_VEL
LIN {X 0,Y 375.976,Z 205.274,A -85,B 0,C 180,E1 -12471.73,E2 -12471.73} C_VEL
LIN {X 0,Y 376.021,Z 205.44,A -85,B 0,C 180,E1 -12474.824,E2 -12474.824} C_VEL
LIN {X 0,Y 379.593,Z 218.477,A -85,B 0,C 180,E1 -12478.038,E2 -12478.038} C_VEL
LIN {X 0,Y 382.563,Z 230.815,A -85,B 0,C 180,E1 -12480.868,E2 -12480.868} C_VEL
LIN {X 0,Y 383.925,Z 236.988,A -85,B 0,C 180,E1 -12482.224,E2 -12482.224} C_VEL
LIN {X 0,Y 383.317,Z 244.616,A -85,B 0,C 180,E1 -12483.632,E2 -12483.632} C_VEL
LIN {X 0,Y 389.277,Z 273.288,A -85,B 0,C 180,E1 -12484.668,E2 -12484.668} C_VEL
LIN {X 0,Y 390.103,Z 277.761,A -85,B 0,C 180,E1 -12484.815,E2 -12484.815} C_VEL
LIN {X 0,Y 388.104,Z 387.984,A -85,B 0,C 180,E1 -12486.77,E2 -12486.77} C_VEL
LIN {X 0,Y 387.448,Z 402.255,A -85,B 0,C 180,E1 -12487.222,E2 -12487.222} C_VEL
LIN {X 0,Y 386.554,Z 416.663,A -85,B 0,C 180,E1 -12487.911,E2 -12487.911} C_VEL
LIN {X 0,Y 385.382,Z 429.759,A -85,B 0,C 180,E1 -12488.749,E2 -12488.749} C_VEL
LIN {X 0,Y 384.144,Z 442.461,A -85,B 0,C 180,E1 -12489.798,E2 -12489.798} C_VEL
LIN {X 0,Y 382.644,Z 454.022,A -85,B 0,C 180,E1 -12490.973,E2 -12490.973} C_VEL
LIN {X 0,Y 381.311,Z 464.603,A -85,B 0,C 180,E1 -12492.295,E2 -12492.295} C_VEL
LIN {X 0,Y 379.769,Z 475.1,A -85,B 0,C 180,E1 -12493.883,E2 -12493.883} C_VEL
LIN {X 0,Y 378.624,Z 483.774,A -85,B 0,C 180,E1 -12495.488,E2 -12495.488} C_VEL
LIN {X 0,Y 377.325,Z 492.112,A -85,B 0,C 180,E1 -12497.358,E2 -12497.358} C_VEL
LIN {X 0,Y 376.417,Z 498.857,A -85,B 0,C 180,E1 -12499.239,E2 -12499.239} C_VEL
LIN {X 0,Y 375.645,Z 504.939,A -85,B 0,C 180,E1 -12501.392,E2 -12501.392} C_VEL
LIN {X 0,Y 375.19,Z 509.476,A -85,B 0,C 180,E1 -12503.547,E2 -12503.547} C_VEL
LIN {X 0,Y 374.794,Z 512.628,A -85,B 0,C 180,E1 -12505.698,E2 -12505.698} C_VEL
LIN {X 0,Y 374.751,Z 514.485,A -85,B 0,C 180,E1 -12507.85,E2 -12507.85} C_VEL
LIN {X 0,Y 374.611,Z 515.123,A -85,B 0,C 180,E1 -12510,E2 -12510} C_VEL
LIN {X 0,Y 374.725,Z 514.544,A -85,B 0,C 180,E1 -12512.149,E2 -12512.149} C_VEL
LIN {X 0,Y 374.776,Z 512.749,A -85,B 0,C 180,E1 -12514.301,E2 -12514.301} C_VEL
LIN {X 0,Y 375.169,Z 509.661,A -85,B 0,C 180,E1 -12516.453,E2 -12516.453} C_VEL
LIN {X 0,Y 375.564,Z 505.277,A -85,B 0,C 180,E1 -12518.573,E2 -12518.573} C_VEL
LIN {X 0,Y 375.159,Z 503.29,A -85,B 0,C 180,E1 -12519.421,E2 -12519.421} C_VEL
LIN {X 0,Y 372.835,Z 499.728,A -85,B 0,C 180,E1 -12520.795,E2 -12520.795} C_VEL
LIN {X 0,Y 370.618,Z 495.571,A -85,B 0,C 180,E1 -12522.143,E2 -12522.143} C_VEL
LIN {X 0,Y 370.385,Z 492.651,A -85,B 0,C 180,E1 -12522.939,E2 -12522.939} C_VEL
LIN {X 0,Y 371.691,Z 484.625,A -85,B 0,C 180,E1 -12524.788,E2 -12524.788} C_VEL
LIN {X 0,Y 372.866,Z 476.062,A -85,B 0,C 180,E1 -12526.422,E2 -12526.422} C_VEL
LIN {X 0,Y 374.495,Z 465.695,A -85,B 0,C 180,E1 -12528.037,E2 -12528.037} C_VEL
LIN {X 0,Y 375.902,Z 455.274,A -85,B 0,C 180,E1 -12529.381,E2 -12529.381} C_VEL
LIN {X 0,Y 377.365,Z 443.943,A -85,B 0,C 180,E1 -12530.58,E2 -12530.58} C_VEL
LIN {X 0,Y 378.715,Z 431.545,A -85,B 0,C 180,E1 -12531.643,E2 -12531.643} C_VEL
LIN {X 0,Y 379.933,Z 417.867,A -85,B 0,C 180,E1 -12532.558,E2 -12532.558} C_VEL
LIN {X 0,Y 380.927,Z 403.649,A -85,B 0,C 180,E1 -12533.261,E2 -12533.261} C_VEL
LIN {X 0,Y 381.611,Z 390.031,A -85,B 0,C 180,E1 -12533.721,E2 -12533.721} C_VEL
LIN {X 0,Y 382.202,Z 366.031,A -85,B 0,C 180,E1 -12534.186,E2 -12534.186} C_VEL
LIN {X 0,Y 383.657,Z 277.907,A -85,B 0,C 180,E1 -12535.769,E2 -12535.769} C_VEL
LIN {X 0,Y 377.976,Z 250.201,A -85,B 0,C 180,E1 -12536.769,E2 -12536.769} C_VEL
LIN {X 0,Y 376.804,Z 244.361,A -85,B 0,C 180,E1 -12537.024,E2 -12537.024} C_VEL
LIN {X 0,Y 377.192,Z 239.324,A -85,B 0,C 180,E1 -12537.983,E2 -12537.983} C_VEL
LIN {X 0,Y 374.502,Z 227.127,A -85,B 0,C 180,E1 -12540.755,E2 -12540.755} C_VEL
LIN {X 0,Y 371.442,Z 215.091,A -85,B 0,C 180,E1 -12543.641,E2 -12543.641} C_VEL
LIN {X 0,Y 368.932,Z 206.262,A -85,B 0,C 180,E1 -12545.927,E2 -12545.927} C_VEL
LIN {X 0,Y 368.901,Z 206.151,A -85,B 0,C 180,E1 -12548.952,E2 -12548.952} C_VEL
LIN {X 0,Y 368.878,Z 206.151,A -85,B 0,C 180,E1 -12552.008,E2 -12552.008} C_VEL
LIN {X 0,Y 368.877,Z 206.152,A -85,B 0,C 180,E1 -12555.175,E2 -12555.175} C_VEL
LIN {X 0,Y 368.879,Z 206.162,A -85,B 0,C 180,E1 -12558.177,E2 -12558.177} C_VEL
LIN {X 0,Y 368.904,Z 206.149,A -85,B 0,C 180,E1 -12561.359,E2 -12561.359} C_VEL
LIN {X 0,Y 368.932,Z 206.135,A -85,B 0,C 180,E1 -12565.146,E2 -12565.146} C_VEL
LIN {X 0,Y 368.924,Z 206.152,A -85,B 0,C 180,E1 -12569.046,E2 -12569.046} C_VEL
LIN {X 0,Y 368.981,Z 206.123,A -85,B 0,C 180,E1 -12571.564,E2 -12571.564} C_VEL
LIN {X 0,Y 368.952,Z 206.15,A -85,B 0,C 180,E1 -12575.224,E2 -12575.224} C_VEL
LIN {X 0,Y 368.932,Z 206.152,A -85,B 0,C 180,E1 -12578.973,E2 -12578.973} C_VEL
LIN {X 0,Y 368.984,Z 206.147,A -85,B 0,C 180,E1 -12582.257,E2 -12582.257} C_VEL
LIN {X 0,Y 369.031,Z 206.142,A -85,B 0,C 180,E1 -12586.227,E2 -12586.227} C_VEL
LIN {X 0,Y 369.061,Z 206.137,A -85,B 0,C 180,E1 -12590.131,E2 -12590.131} C_VEL
LIN {X 0,Y 369.181,Z 206.116,A -85,B 0,C 180,E1 -12592.342,E2 -12592.342} C_VEL
LIN {X 0,Y 369.138,Z 206.131,A -85,B 0,C 180,E1 -12594.537,E2 -12594.537} C_VEL
LIN {X 0,Y 369.312,Z 206.101,A -85,B 0,C 180,E1 -12597.819,E2 -12597.819} C_VEL
LIN {X 0,Y 369.451,Z 206.089,A -85,B 0,C 180,E1 -12600,E2 -12600} C_VEL
LIN {X 0,Y 369.312,Z 206.101,A -85,B 0,C 180,E1 -12602.181,E2 -12602.181} C_VEL
LIN {X 0,Y 369.201,Z 206.118,A -85,B 0,C 180,E1 -12606.558,E2 -12606.558} C_VEL
LIN {X 0,Y 369.13,Z 206.124,A -85,B 0,C 180,E1 -12608.761,E2 -12608.761} C_VEL
LIN {X 0,Y 368.999,Z 206.148,A -85,B 0,C 180,E1 -12612.093,E2 -12612.093} C_VEL
LIN {X 0,Y 368.991,Z 206.145,A -85,B 0,C 180,E1 -12615.465,E2 -12615.465} C_VEL
LIN {X 0,Y 368.976,Z 206.146,A -85,B 0,C 180,E1 -12618.893,E2 -12618.893} C_VEL
LIN {X 0,Y 368.926,Z 206.155,A -85,B 0,C 180,E1 -12622.395,E2 -12622.395} C_VEL
LIN {X 0,Y 368.993,Z 206.121,A -85,B 0,C 180,E1 -12625.98,E2 -12625.98} C_VEL
LIN {X 0,Y 368.955,Z 206.148,A -85,B 0,C 180,E1 -12628.812,E2 -12628.812} C_VEL
LIN {X 0,Y 368.892,Z 206.137,A -85,B 0,C 180,E1 -12632.238,E2 -12632.238} C_VEL
LIN {X 0,Y 368.923,Z 206.155,A -85,B 0,C 180,E1 -12635.002,E2 -12635.002} C_VEL
LIN {X 0,Y 368.903,Z 206.149,A -85,B 0,C 180,E1 -12638.641,E2 -12638.641} C_VEL
LIN {X 0,Y 368.875,Z 206.148,A -85,B 0,C 180,E1 -12642.01,E2 -12642.01} C_VEL
LIN {X 0,Y 368.874,Z 206.152,A -85,B 0,C 180,E1 -12645.176,E2 -12645.176} C_VEL
LIN {X 0,Y 368.87,Z 206.147,A -85,B 0,C 180,E1 -12648.177,E2 -12648.177} C_VEL
LIN {X 0,Y 368.942,Z 206.161,A -85,B 0,C 180,E1 -12651.925,E2 -12651.925} C_VEL
LIN {X 0,Y 368.972,Z 206.502,A -85,B 0,C 180,E1 -12652.188,E2 -12652.188} C_VEL
LIN {X 0,Y 372.787,Z 219.064,A -85,B 0,C 180,E1 -12655.054,E2 -12655.054} C_VEL
LIN {X 0,Y 376.531,Z 232.743,A -85,B 0,C 180,E1 -12657.939,E2 -12657.939} C_VEL
LIN {X 0,Y 378.92,Z 242.893,A -85,B 0,C 180,E1 -12659.949,E2 -12659.949} C_VEL
LIN {X 0,Y 378.908,Z 245.07,A -85,B 0,C 180,E1 -12660.295,E2 -12660.295} C_VEL
LIN {X 0,Y 383.096,Z 270.134,A -85,B 0,C 180,E1 -12661.194,E2 -12661.194} C_VEL
LIN {X 0,Y 384.364,Z 279.015,A -85,B 0,C 180,E1 -12661.482,E2 -12661.482} C_VEL
LIN {X 0,Y 381.102,Z 406.402,A -85,B 0,C 180,E1 -12664.026,E2 -12664.026} C_VEL
LIN {X 0,Y 380.219,Z 422.094,A -85,B 0,C 180,E1 -12664.549,E2 -12664.549} C_VEL
LIN {X 0,Y 379.048,Z 436.888,A -85,B 0,C 180,E1 -12665.256,E2 -12665.256} C_VEL
LIN {X 0,Y 377.726,Z 450.763,A -85,B 0,C 180,E1 -12666.13,E2 -12666.13} C_VEL
LIN {X 0,Y 376.231,Z 464.172,A -85,B 0,C 180,E1 -12667.195,E2 -12667.195} C_VEL
LIN {X 0,Y 374.537,Z 477.791,A -85,B 0,C 180,E1 -12668.537,E2 -12668.537} C_VEL
LIN {X 0,Y 373.108,Z 489.149,A -85,B 0,C 180,E1 -12669.894,E2 -12669.894} C_VEL
LIN {X 0,Y 371.772,Z 500.605,A -85,B 0,C 180,E1 -12671.541,E2 -12671.541} C_VEL
LIN {X 0,Y 370.317,Z 511.685,A -85,B 0,C 180,E1 -12673.461,E2 -12673.461} C_VEL
LIN {X 0,Y 369.234,Z 520.88,A -85,B 0,C 180,E1 -12675.393,E2 -12675.393} C_VEL
LIN {X 0,Y 368.501,Z 528.523,A -85,B 0,C 180,E1 -12677.331,E2 -12677.331} C_VEL
LIN {X 0,Y 367.859,Z 535.591,A -85,B 0,C 180,E1 -12679.543,E2 -12679.543} C_VEL
LIN {X 0,Y 367.579,Z 541.121,A -85,B 0,C 180,E1 -12681.756,E2 -12681.756} C_VEL
LIN {X 0,Y 367.488,Z 545.254,A -85,B 0,C 180,E1 -12683.971,E2 -12683.971} C_VEL
LIN {X 0,Y 367.443,Z 547.441,A -85,B 0,C 180,E1 -12685.613,E2 -12685.613} C_VEL
LIN {X 0,Y 367.484,Z 549.312,A -85,B 0,C 180,E1 -12687.808,E2 -12687.808} C_VEL
LIN {X 0,Y 367.539,Z 549.947,A -85,B 0,C 180,E1 -12690,E2 -12690} C_VEL
LIN {X 0,Y 367.484,Z 549.305,A -85,B 0,C 180,E1 -12692.192,E2 -12692.192} C_VEL
LIN {X 0,Y 367.477,Z 547.426,A -85,B 0,C 180,E1 -12694.388,E2 -12694.388} C_VEL
LIN {X 0,Y 367.549,Z 544.288,A -85,B 0,C 180,E1 -12696.588,E2 -12696.588} C_VEL
LIN {X 0,Y 367.626,Z 539.814,A -85,B 0,C 180,E1 -12698.798,E2 -12698.798} C_VEL
LIN {X 0,Y 368.023,Z 533.903,A -85,B 0,C 180,E1 -12701.009,E2 -12701.009} C_VEL
LIN {X 0,Y 368.676,Z 526.397,A -85,B 0,C 180,E1 -12703.224,E2 -12703.224} C_VEL
LIN {X 0,Y 369.536,Z 518.338,A -85,B 0,C 180,E1 -12705.16,E2 -12705.16} C_VEL
LIN {X 0,Y 370.662,Z 508.628,A -85,B 0,C 180,E1 -12707.091,E2 -12707.091} C_VEL
LIN {X 0,Y 372.111,Z 497.293,A -85,B 0,C 180,E1 -12708.95,E2 -12708.95} C_VEL
LIN {X 0,Y 373.508,Z 485.797,A -85,B 0,C 180,E1 -12710.515,E2 -12710.515} C_VEL
LIN {X 0,Y 375.024,Z 473.82,A -85,B 0,C 180,E1 -12711.868,E2 -12711.868} C_VEL
LIN {X 0,Y 376.588,Z 460.846,A -85,B 0,C 180,E1 -12713.073,E2 -12713.073} C_VEL
LIN {X 0,Y 378.129,Z 446.631,A -85,B 0,C 180,E1 -12714.136,E2 -12714.136} C_VEL
LIN {X 0,Y 379.361,Z 432.5,A -85,B 0,C 180,E1 -12714.964,E2 -12714.964} C_VEL
LIN {X 0,Y 380.466,Z 417.397,A -85,B 0,C 180,E1 -12715.618,E2 -12715.618} C_VEL
LIN {X 0,Y 381.25,Z 401.563,A -85,B 0,C 180,E1 -12716.074,E2 -12716.074} C_VEL
LIN {X 0,Y 384.318,Z 278.65,A -85,B 0,C 180,E1 -12718.514,E2 -12718.514} C_VEL
LIN {X 0,Y 379.37,Z 247.943,A -85,B 0,C 180,E1 -12719.567,E2 -12719.567} C_VEL
LIN {X 0,Y 378.919,Z 244.823,A -85,B 0,C 180,E1 -12719.716,E2 -12719.716} C_VEL
LIN {X 0,Y 378.575,Z 241.396,A -85,B 0,C 180,E1 -12720.329,E2 -12720.329} C_VEL
LIN {X 0,Y 375.465,Z 228.768,A -85,B 0,C 180,E1 -12722.876,E2 -12722.876} C_VEL
LIN {X 0,Y 371.853,Z 215.88,A -85,B 0,C 180,E1 -12725.64,E2 -12725.64} C_VEL
LIN {X 0,Y 368.939,Z 206.262,A -85,B 0,C 180,E1 -12727.882,E2 -12727.882} C_VEL
LIN {X 0,Y 368.904,Z 206.119,A -85,B 0,C 180,E1 -12730.371,E2 -12730.371} C_VEL
LIN {X 0,Y 368.881,Z 206.155,A -85,B 0,C 180,E1 -12733.616,E2 -12733.616} C_VEL
LIN {X 0,Y 368.884,Z 206.157,A -85,B 0,C 180,E1 -12736.696,E2 -12736.696} C_VEL
LIN {X 0,Y 368.91,Z 206.158,A -85,B 0,C 180,E1 -12739.643,E2 -12739.643} C_VEL
LIN {X 0,Y 368.9,Z 206.148,A -85,B 0,C 180,E1 -12743.144,E2 -12743.144} C_VEL
LIN {X 0,Y 368.895,Z 206.144,A -85,B 0,C 180,E1 -12746.462,E2 -12746.462} C_VEL
LIN {X 0,Y 368.927,Z 206.149,A -85,B 0,C 180,E1 -12749.047,E2 -12749.047} C_VEL
LIN {X 0,Y 368.978,Z 206.143,A -85,B 0,C 180,E1 -12751.564,E2 -12751.564} C_VEL
LIN {X 0,Y 368.998,Z 206.12,A -85,B 0,C 180,E1 -12754.02,E2 -12754.02} C_VEL
LIN {X 0,Y 368.93,Z 206.154,A -85,B 0,C 180,E1 -12757.605,E2 -12757.605} C_VEL
LIN {X 0,Y 368.98,Z 206.145,A -85,B 0,C 180,E1 -12761.107,E2 -12761.107} C_VEL
LIN {X 0,Y 368.996,Z 206.145,A -85,B 0,C 180,E1 -12764.535,E2 -12764.535} C_VEL
LIN {X 0,Y 369.003,Z 206.147,A -85,B 0,C 180,E1 -12767.907,E2 -12767.907} C_VEL
LIN {X 0,Y 369.164,Z 206.126,A -85,B 0,C 180,E1 -12771.869,E2 -12771.869} C_VEL
LIN {X 0,Y 369.141,Z 206.119,A -85,B 0,C 180,E1 -12774.538,E2 -12774.538} C_VEL
LIN {X 0,Y 369.314,Z 206.101,A -85,B 0,C 180,E1 -12777.819,E2 -12777.819} C_VEL
LIN {X 0,Y 369.454,Z 206.088,A -85,B 0,C 180,E1 -12780,E2 -12780} C_VEL
LIN {X 0,Y 369.314,Z 206.101,A -85,B 0,C 180,E1 -12782.181,E2 -12782.181} C_VEL
LIN {X 0,Y 369.202,Z 206.116,A -85,B 0,C 180,E1 -12786.616,E2 -12786.616} C_VEL
LIN {X 0,Y 369.136,Z 206.124,A -85,B 0,C 180,E1 -12788.761,E2 -12788.761} C_VEL
LIN {X 0,Y 369.003,Z 206.137,A -85,B 0,C 180,E1 -12792.094,E2 -12792.094} C_VEL
LIN {X 0,Y 368.996,Z 206.139,A -85,B 0,C 180,E1 -12795.465,E2 -12795.465} C_VEL
LIN {X 0,Y 368.957,Z 206.15,A -85,B 0,C 180,E1 -12798.894,E2 -12798.894} C_VEL
LIN {X 0,Y 368.935,Z 206.153,A -85,B 0,C 180,E1 -12802.395,E2 -12802.395} C_VEL
LIN {X 0,Y 368.999,Z 206.144,A -85,B 0,C 180,E1 -12805.98,E2 -12805.98} C_VEL
LIN {X 0,Y 368.914,Z 206.137,A -85,B 0,C 180,E1 -12809.691,E2 -12809.691} C_VEL
LIN {X 0,Y 368.896,Z 206.152,A -85,B 0,C 180,E1 -12813.043,E2 -12813.043} C_VEL
LIN {X 0,Y 368.918,Z 206.148,A -85,B 0,C 180,E1 -12816.197,E2 -12816.197} C_VEL
LIN {X 0,Y 368.902,Z 206.145,A -85,B 0,C 180,E1 -12818.954,E2 -12818.954} C_VEL
LIN {X 0,Y 368.882,Z 206.161,A -85,B 0,C 180,E1 -12822.01,E2 -12822.01} C_VEL
LIN {X 0,Y 368.88,Z 206.155,A -85,B 0,C 180,E1 -12825.176,E2 -12825.176} C_VEL
LIN {X 0,Y 368.883,Z 206.151,A -85,B 0,C 180,E1 -12828.178,E2 -12828.178} C_VEL
LIN {X 0,Y 368.91,Z 206.15,A -85,B 0,C 180,E1 -12831.36,E2 -12831.36} C_VEL
LIN {X 0,Y 368.956,Z 206.38,A -85,B 0,C 180,E1 -12834.238,E2 -12834.238} C_VEL
LIN {X 0,Y 372.14,Z 217.712,A -85,B 0,C 180,E1 -12837.115,E2 -12837.115} C_VEL
LIN {X 0,Y 375.082,Z 229.418,A -85,B 0,C 180,E1 -12839.901,E2 -12839.901} C_VEL
LIN {X 0,Y 377.157,Z 238.816,A -85,B 0,C 180,E1 -12842.021,E2 -12842.021} C_VEL
LIN {X 0,Y 376.76,Z 244.523,A -85,B 0,C 180,E1 -12843.095,E2 -12843.095} C_VEL
LIN {X 0,Y 383.107,Z 275.186,A -85,B 0,C 180,E1 -12844.239,E2 -12844.239} C_VEL
LIN {X 0,Y 383.75,Z 279.178,A -85,B 0,C 180,E1 -12844.366,E2 -12844.366} C_VEL
LIN {X 0,Y 381.666,Z 387.741,A -85,B 0,C 180,E1 -12846.318,E2 -12846.318} C_VEL
LIN {X 0,Y 381.001,Z 402.194,A -85,B 0,C 180,E1 -12846.778,E2 -12846.778} C_VEL
LIN {X 0,Y 380.174,Z 415.478,A -85,B 0,C 180,E1 -12847.409,E2 -12847.409} C_VEL
LIN {X 0,Y 378.945,Z 428.505,A -85,B 0,C 180,E1 -12848.227,E2 -12848.227} C_VEL
LIN {X 0,Y 377.67,Z 441.5,A -85,B 0,C 180,E1 -12849.294,E2 -12849.294} C_VEL
LIN {X 0,Y 376.102,Z 453.283,A -85,B 0,C 180,E1 -12850.487,E2 -12850.487} C_VEL
LIN {X 0,Y 374.845,Z 463.081,A -85,B 0,C 180,E1 -12851.697,E2 -12851.697} C_VEL
LIN {X 0,Y 373.189,Z 473.885,A -85,B 0,C 180,E1 -12853.31,E2 -12853.31} C_VEL
LIN {X 0,Y 371.979,Z 482.819,A -85,B 0,C 180,E1 -12854.942,E2 -12854.942} C_VEL
LIN {X 0,Y 370.57,Z 491.383,A -85,B 0,C 180,E1 -12856.845,E2 -12856.845} C_VEL
LIN {X 0,Y 369.687,Z 497.454,A -85,B 0,C 180,E1 -12858.485,E2 -12858.485} C_VEL
LIN {X 0,Y 368.797,Z 503.909,A -85,B 0,C 180,E1 -12860.678,E2 -12860.678} C_VEL
LIN {X 0,Y 368.237,Z 508.946,A -85,B 0,C 180,E1 -12862.956,E2 -12862.956} C_VEL
LIN {X 0,Y 367.913,Z 511.554,A -85,B 0,C 180,E1 -12864.519,E2 -12864.519} C_VEL
LIN {X 0,Y 367.694,Z 514.046,A -85,B 0,C 180,E1 -12866.712,E2 -12866.712} C_VEL
LIN {X 0,Y 367.579,Z 515.288,A -85,B 0,C 180,E1 -12868.904,E2 -12868.904} C_VEL
LIN {X 0,Y 367.577,Z 515.316,A -85,B 0,C 180,E1 -12871.095,E2 -12871.095} C_VEL
LIN {X 0,Y 367.685,Z 514.134,A -85,B 0,C 180,E1 -12873.287,E2 -12873.287} C_VEL
LIN {X 0,Y 367.901,Z 511.705,A -85,B 0,C 180,E1 -12875.48,E2 -12875.48} C_VEL
LIN {X 0,Y 368.321,Z 507.947,A -85,B 0,C 180,E1 -12877.675,E2 -12877.675} C_VEL
LIN {X 0,Y 368.955,Z 502.735,A -85,B 0,C 180,E1 -12879.871,E2 -12879.871} C_VEL
LIN {X 0,Y 369.925,Z 495.894,A -85,B 0,C 180,E1 -12882.062,E2 -12882.062} C_VEL
LIN {X 0,Y 370.385,Z 492.651,A -85,B 0,C 180,E1 -12882.939,E2 -12882.939} C_VEL
LIN {X 0,Y 370.188,Z 489.629,A -85,B 0,C 180,E1 -12883.72,E2 -12883.72} C_VEL
LIN {X 0,Y 368.205,Z 484.475,A -85,B 0,C 180,E1 -12885.003,E2 -12885.003} C_VEL
LIN {X 0,Y 366.323,Z 478.933,A -85,B 0,C 180,E1 -12886.25,E2 -12886.25} C_VEL
LIN {X 0,Y 366.277,Z 475.133,A -85,B 0,C 180,E1 -12886.961,E2 -12886.961} C_VEL
LIN {X 0,Y 367.761,Z 466.081,A -85,B 0,C 180,E1 -12888.379,E2 -12888.379} C_VEL
LIN {X 0,Y 369.24,Z 455.681,A -85,B 0,C 180,E1 -12889.745,E2 -12889.745} C_VEL
LIN {X 0,Y 370.754,Z 444.382,A -85,B 0,C 180,E1 -12890.964,E2 -12890.964} C_VEL
LIN {X 0,Y 372.149,Z 432.03,A -85,B 0,C 180,E1 -12892.044,E2 -12892.044} C_VEL
LIN {X 0,Y 373.459,Z 418.136,A -85,B 0,C 180,E1 -12892.99,E2 -12892.99} C_VEL
LIN {X 0,Y 374.453,Z 404.332,A -85,B 0,C 180,E1 -12893.688,E2 -12893.688} C_VEL
LIN {X 0,Y 375.163,Z 390.972,A -85,B 0,C 180,E1 -12894.154,E2 -12894.154} C_VEL
LIN {X 0,Y 375.684,Z 371.266,A -85,B 0,C 180,E1 -12894.559,E2 -12894.559} C_VEL
LIN {X 0,Y 377.357,Z 279.079,A -85,B 0,C 180,E1 -12896.238,E2 -12896.238} C_VEL
LIN {X 0,Y 371.504,Z 250.545,A -85,B 0,C 180,E1 -12897.299,E2 -12897.299} C_VEL
LIN {X 0,Y 370.226,Z 244.479,A -85,B 0,C 180,E1 -12897.565,E2 -12897.565} C_VEL
LIN {X 0,Y 370.467,Z 242.061,A -85,B 0,C 180,E1 -12898.003,E2 -12898.003} C_VEL
LIN {X 0,Y 368.821,Z 233.498,A -85,B 0,C 180,E1 -12899.947,E2 -12899.947} C_VEL
LIN {X 0,Y 365.825,Z 221.356,A -85,B 0,C 180,E1 -12902.868,E2 -12902.868} C_VEL
LIN {X 0,Y 362.924,Z 210.71,A -85,B 0,C 180,E1 -12905.577,E2 -12905.577} C_VEL
LIN {X 0,Y 361.883,Z 207.12,A -85,B 0,C 180,E1 -12906.58,E2 -12906.58} C_VEL
LIN {X 0,Y 361.853,Z 207.031,A -85,B 0,C 180,E1 -12909.86,E2 -12909.86} C_VEL
LIN {X 0,Y 361.833,Z 207.029,A -85,B 0,C 180,E1 -12912.828,E2 -12912.828} C_VEL
LIN {X 0,Y 361.814,Z 207.028,A -85,B 0,C 180,E1 -12915.946,E2 -12915.946} C_VEL
LIN {X 0,Y 361.831,Z 207.028,A -85,B 0,C 180,E1 -12919.244,E2 -12919.244} C_VEL
LIN {X 0,Y 361.86,Z 207.038,A -85,B 0,C 180,E1 -12922.776,E2 -12922.776} C_VEL
LIN {X 0,Y 361.851,Z 207.017,A -85,B 0,C 180,E1 -12925.719,E2 -12925.719} C_VEL
LIN {X 0,Y 361.872,Z 207.023,A -85,B 0,C 180,E1 -12929.672,E2 -12929.672} C_VEL
LIN {X 0,Y 361.95,Z 207.019,A -85,B 0,C 180,E1 -12933.474,E2 -12933.474} C_VEL
LIN {X 0,Y 361.884,Z 207.029,A -85,B 0,C 180,E1 -12937.144,E2 -12937.144} C_VEL
LIN {X 0,Y 361.915,Z 207.022,A -85,B 0,C 180,E1 -12940.724,E2 -12940.724} C_VEL
LIN {X 0,Y 361.94,Z 207.016,A -85,B 0,C 180,E1 -12944.226,E2 -12944.226} C_VEL
LIN {X 0,Y 361.993,Z 207.021,A -85,B 0,C 180,E1 -12946.527,E2 -12946.527} C_VEL
LIN {X 0,Y 362.025,Z 207.013,A -85,B 0,C 180,E1 -12949.938,E2 -12949.938} C_VEL
LIN {X 0,Y 362.144,Z 206.993,A -85,B 0,C 180,E1 -12952.192,E2 -12952.192} C_VEL
LIN {X 0,Y 362.111,Z 207.005,A -85,B 0,C 180,E1 -12954.431,E2 -12954.431} C_VEL
LIN {X 0,Y 362.276,Z 206.977,A -85,B 0,C 180,E1 -12957.776,E2 -12957.776} C_VEL
LIN {X 0,Y 362.421,Z 206.964,A -85,B 0,C 180,E1 -12960,E2 -12960} C_VEL
LIN {X 0,Y 362.276,Z 206.978,A -85,B 0,C 180,E1 -12962.223,E2 -12962.223} C_VEL
LIN {X 0,Y 362.165,Z 206.996,A -85,B 0,C 180,E1 -12966.686,E2 -12966.686} C_VEL
LIN {X 0,Y 362.067,Z 207.003,A -85,B 0,C 180,E1 -12968.933,E2 -12968.933} C_VEL
LIN {X 0,Y 361.953,Z 207.022,A -85,B 0,C 180,E1 -12972.332,E2 -12972.332} C_VEL
LIN {X 0,Y 361.955,Z 207.02,A -85,B 0,C 180,E1 -12974.62,E2 -12974.62} C_VEL
LIN {X 0,Y 361.953,Z 207.017,A -85,B 0,C 180,E1 -12978.099,E2 -12978.099} C_VEL
LIN {X 0,Y 361.885,Z 207.026,A -85,B 0,C 180,E1 -12981.653,E2 -12981.653} C_VEL
LIN {X 0,Y 361.922,Z 207.01,A -85,B 0,C 180,E1 -12985.29,E2 -12985.29} C_VEL
LIN {X 0,Y 361.912,Z 207.01,A -85,B 0,C 180,E1 -12987.779,E2 -12987.779} C_VEL
LIN {X 0,Y 361.84,Z 207.024,A -85,B 0,C 180,E1 -12991.286,E2 -12991.286} C_VEL
LIN {X 0,Y 361.848,Z 207.033,A -85,B 0,C 180,E1 -12994.281,E2 -12994.281} C_VEL
